# B&R Automation Studio project x20ost (part 3)

#### bnrdirmodule.c
```c
/********************************************************************
 * COPYRIGHT -- Kontora
 ********************************************************************
 * Program: bnrmain
 * File: bnrlsens.c
 * Author: Abramenya
 * Created: January 19, 2009
 *******************************************************************/

#include "bnrdirmodule.h"
#ifdef _DEFAULT_INCLUDES
 #include <AsDefault.h>
#endif
#if MYSYSTEM_ID != 5
void CDirectionModule_Init(This,SDIRTABLE *pDirect,CMFlash *pFlash)
{
    DECLARE_SINGLE_OPEN(CDirectionModule)
	INT i,nCreated;
	BOOL blSerialize;
	BYTE bySensorType,byLen;
	CSensor *pSensor;
	CSmartSensor *pSmartSensor;
	CIdleSensor *pIdleSensor;
	CDigitalSensor *pDgSensor;
	SNSPARAMTABLE *sP;
	pT->m_pDirTable = pDirect;
	pT->m_pFlash = pFlash;
	pT->m_wSensorMode = 0;
	pT->m_pvInGate = pDirect->pvIn;
	pT->m_pvOutGate = pDirect->pvOut;
	pT->m_byDefSett = 0;
    #if MYSYSTEM_ID == 4
	pT->m_byAmInpGate = ((SDIGGATES*)pT->m_pvInGate)->byAmGate;
    #else
    pT->m_byAmInpGate = ((SINPUTGATE*)pT->m_pvInGate)->byAmInGate;
    #endif
	pT->m_wLayerMode  = 0x2;
	/*
	#if   MYSYSTEM_ID == 0
	 pT->m_wLayerMode  = 0x2;
	#elif MYSYSTEM_ID == 1
	 pT->m_wLayerMode  = 0x1;
	#elif MYSYSTEM_ID == 2
	 pT->m_wLayerMode  = 0x2;
	#elif MYSYSTEM_ID == 3
	 pT->m_wLayerMode  = 0x1a;
	#endif
	*/
	pT->m_blGetData = FALSE;
    #ifdef DEB_CDirectionModule
	Info("\n(%b)CDIRC::>Create Direction.",&pDirect->byDirectionID);
    #endif
	pT->m_byStatSnsConn = 0xff;
	pT->m_byDirectionID = pDirect->byDirectionID;
	pT->m_byAmSwitching = pDirect->byAmSwitching;
	pT->m_byDirectionCode = pDirect->byDirectionCode;
    New(sizeof(CSensor*)*pT->m_byAmSwitching,pT->m_pSensor);
	for (i=0;i<pT->m_byAmSwitching;i++)pT->m_pSensor[i]=0;
	for (nCreated=0;nCreated<=1;nCreated++)
	{
	if(nCreated)
	{
     #if MYSYSTEM_ID != 4
	 pT->SetInputGate(pT,pT->m_pvInGate);
     #endif
	 blSerialize = pT->Serialize(pT,FALSE);
	}
	for (i=0;i<pT->m_byAmSwitching;i++)
	{
	 bySensorType = pDirect->sSwitchTable[i].bySwitchCommand;
	 switch(bySensorType)
	 {
	    case SWC_CMD_SMR_CON:
			{
			 if(nCreated==0){
			 New(sizeof(CSmartSensor),pSmartSensor);
			 InitObject(CSmartSensor,pSmartSensor);
			 pSmartSensor->pBase->m_bySystemID = pT->m_bySystemID;
			 pT->m_pSensor[i] = pSmartSensor->pBase;}
			 if(nCreated==1){
			 pSmartSensor->pBase = pT->m_pSensor[i];
			 pT->SwitchSensor(pT,pSmartSensor->pBase,&pDirect->sSwitchTable[i]);
			 pSmartSensor->pBase->SetDirection(pSmartSensor->pBase,pT,pT->m_byDirectionID);
			 pSmartSensor->pBase->Init(pSmartSensor->pBase,&pDirect->sSwitchTable[i]);}
			}
		break;
		case SWC_CMD_IDL_CON:
			{
			 if(nCreated==0){
			 New(sizeof(CIdleSensor),pIdleSensor);
			 InitObject(CIdleSensor,pIdleSensor);
			 pIdleSensor->pBase->m_bySystemID = pT->m_bySystemID;
			 pT->m_pSensor[i] = pIdleSensor->pBase;}
			 if(nCreated==1){
			 pIdleSensor->pBase = pT->m_pSensor[i];
			 pT->SwitchSensor(pT,pIdleSensor->pBase,&pDirect->sSwitchTable[i]);
			 pIdleSensor->pBase->SetDirection(pIdleSensor->pBase,pT,pT->m_byDirectionID);
			 pIdleSensor->pBase->Init(pIdleSensor->pBase,&pDirect->sSwitchTable[i]);}
			}
		break;
		case SWC_CMD_EMT_CON:
			{
			 if(nCreated==0){
			 New(sizeof(CSensor),pSensor);
			 InitObject(CSensor,pSensor);
			 pSensor->m_bySystemID = pT->m_bySystemID;
			 pT->m_pSensor[i] = pSensor;}
			 if(nCreated==1){
			 pSensor->pBase = pT->m_pSensor[i];
			 pSensor->SetDirection(pSensor,pT,pT->m_byDirectionID);
			 pSensor->Init(pSensor,&pDirect->sSwitchTable[i]);}
			}
		break;
		case SWC_CMD_LOG_CON:
			{
			 if(nCreated==0){
			 New(sizeof(CDigitalSensor),pDgSensor);
			 InitObject(CDigitalSensor,pDgSensor);
			 pDgSensor->pBase->m_bySystemID = pT->m_bySystemID;
			 pT->m_pSensor[i] = pDgSensor->pBase;}
			 if(nCreated==1){
			 pDgSensor->pBase = pT->m_pSensor[i];
             pDgSensor->pBase->SetDirection(pDgSensor->pBase,pT,pT->m_byDirectionID);
			 pDgSensor->pBase->InitDigital(pDgSensor->pBase,&pDirect->sSwitchTable[i]);//Create In Out
			 pT->SwitchDigitalSensor(pT,pDgSensor->pBase,&pDirect->sSwitchTable[i]);}   //Connect In or Out
			}
		break;
		default:
		break;
	 }
	}
	}
    #if MYSYSTEM_ID != 4
	if (blSerialize)for(i=0;i<8;i++)if(pT->m_nST.m_wLayerMode&(1<<i))pT->SetCurentTank(pT,i);
    #endif
}
BOOL CDirectionModule_EventHandler(This,SMESSAGE *pMsg)
{
    DECLARE_SINGLE_OPEN(CDirectionModule)
	INT16 **pwData;
	CSensor *pSN;
	BYTE byParam;
    switch(pMsg->m_sbyFor)
	{
		case MDL_DIRMD:
			 switch(pMsg->m_sbyType)
			 {
			    case EV_DIRMD_SET_TANK_REQ:
	                 pT->SetCurentTank(pT,pMsg->m_sbySensor);
                     #ifdef DEB_CDirectionModule
					 Info("\n(%b)CDIRC::>(%b)(%b)SetTank.",&pT->m_bySystemID,&pT->m_byDirectionID,&pMsg->m_sbySensor);
                     #endif
				break;
				#if MYSYSTEM_ID != 4
			 	case EV_DIRMD_GET_PARAM_REQ:
					 if(pMsg->m_sbySensor<pT->m_byAmSwitching)
					 {
					  pSN = pT->m_pSensor[pMsg->m_sbySensor];
					  byParam = pMsg->m_sbyInfo[1];
					  pSN->GetParamTable(pSN,pMsg->m_sbyInfo[1]);
                      #ifdef DEB_CDirectionModule
					  Info("\n(%b)CDIRC::>(%b)(%b)GetParam.",&pT->m_bySystemID,&pT->m_byDirectionID,&pMsg->m_sbySensor);
                      #endif
					 }
				break;
				case EV_DIRMD_CONN_STAT_SNS_IND:
                     #ifdef DEB_CDirectionModule
					 Info("\n(%b)CDIRC::>(%b)(%b)Connect To Sensor.",&pT->m_bySystemID,&pT->m_byDirectionID,&pMsg->m_sbySensor);
                     #endif
					 pT->m_byStatSnsConn  = pMsg->m_sbySensor;
					 pT->m_byTypeTest     = 0;
					 if(pMsg->m_sbySensor<pT->m_byAmSwitching)
					 {
					  pSN = pT->m_pSensor[pMsg->m_sbySensor];
					  pT->m_pStatSnsTmr.SetTimer(&pT->m_pStatSnsTmr,MDL_DIRMD,MDL_DIRMD,EV_DIRMD_REFR_TIM_PROC_IND,pSN->m_byDirection,0,DEV_SYSTM_BOX_ID);
					  pSN->GetParamTable(pSN,MDL_TPIDT);
					 }
				break;
			    case EV_DIRMD_DISC_STAT_SNS_IND:
                     #ifdef DEB_CDirectionModule
					 Info("\n(%b)CDIRC::>(%b)Disconnect To Sensor.",&pT->m_bySystemID,&pT->m_byDirectionID);
                     #endif
					 pT->m_byStatSnsConn = 0xff;
				break;
                #endif
			    case EV_DIRMD_CONN_STAT_START_IND:
                     #ifdef DEB_CDirectionModule
					 Info("\n(%b)CDIRC::>(%b)(%b)Start Stat Proc:%b.",&pT->m_bySystemID,&pT->m_byDirectionID,&pMsg->m_sbySensor,&pMsg->m_sbyInfo[1]);
                     #endif
					 if((pMsg->m_sbySensor<pT->m_byAmSwitching)&&(pT->m_byStatSnsConn!=0xff))
					 {
					  pSN = pT->m_pSensor[pMsg->m_sbySensor];
					  pT->m_byTypeTest = pMsg->m_sbyInfo[2];
					  if(pT->m_byTypeTest==0)pSN->StartCaptureProc(pSN);
					  pT->m_pStatSnsTmr.OnTimer(&pT->m_pStatSnsTmr,pMsg->m_sbyInfo[1]*SYSTEM_QTIME/100);
					 }
				break;
			    case EV_DIRMD_CONN_STAT_STOP_IND:
                     #ifdef DEB_CDirectionModule
					 Info("\n(%b)CDIRC::>(%b)(%b)Stop Stat Proc.",&pT->m_bySystemID,&pT->m_byDirectionID,&pMsg->m_sbySensor);
                     #endif
					 if(pMsg->m_sbySensor<pT->m_byAmSwitching)
					 {
					  pSN = pT->m_pSensor[pMsg->m_sbySensor];
 					  pT->m_pStatSnsTmr.OfTimer(&pT->m_pStatSnsTmr);
					 }
			    break;
				case EV_DIRMD_REFR_TIM_PROC_IND:
					 if(pT->m_byStatSnsConn!=0xff)
					 {
					 pMsg->m_sbyFrom      = MDL_DIRMD;
					 pMsg->m_sbyFor       = MDL_TPIDT;
					 pMsg->m_sbyIntType   = DEV_ARM_PORT_TCP;
					 pMsg->m_sbyServerID  = pT->m_bySystemID;
					 pMsg->m_sbyType      = EV_DIRMD_STAT_DATA_IND;
					 pMsg->m_sbyDirection = pT->m_byDirectionID;
	                 pMsg->m_sbySensor    = pT->m_byStatSnsConn;
 				     pSN                  = pT->m_pSensor[pT->m_byStatSnsConn];
                     if(pT->m_byTypeTest==0)
					 {
					  pMsg->m_sbyInfo[0] = (BYTE)pSN->m_wStatIndex;
					  pMsg->m_sbyInfo[1] = (BYTE)pSN->m_wStatIndex;
					  pwData = pSN->GetCaptureBuffer(pSN);
					  memcpy(&pMsg->m_sbyInfo[2],pwData,12*pSN->m_wStatQuant);
					  pMsg->m_swLen = 9+1+1+12*pSN->m_wStatQuant;
					 }
					 if(pT->m_byTypeTest==1)
					 {
					  pSN->CaptureData(pSN->pChld);
					  pwData = pSN->GetCaptureBuffer(pSN);
					  pMsg->m_sbyInfo[0] = (BYTE)pSN->m_wStatIndex;
					  pMsg->m_sbyInfo[1] = (BYTE)pSN->m_wStatIndex;
					  memcpy(&pMsg->m_sbyInfo[2],pwData,4*pSN->m_wStatIndex);
					  pMsg->m_swLen = 9+1+1+4*pSN->m_wStatIndex;
					 }
					 FPUT(DEV_ARMOT_BOX_ID,(BYTE*)&pMsg->m_swLen);
                     if(dwFL&DEB_OUT_OBSR_COMM)
	                 Info("\n(%b)COBSE::>msg:%M",&pT->m_bySystemID,(BYTE*)pMsg);
					 pSN->RestartCaptureProc(pSN);
					 pT->m_pStatSnsTmr.Restart(&pT->m_pStatSnsTmr);
					 }
				break;
			    default:
			    break;
			 }
		break;
		default:
		break;
	}
	return TRUE;
}
void CDirectionModule_SetInputGate(This,SINPUTGATE *pING)
{
    DECLARE_SINGLE_OPEN(CDirectionModule)
	REAL Imin,Imax,R;
	BYTE i;
	CSlot *pSL;
	CPin  *pPN;
	for (i=0;i<pT->m_byAmInpGate;i++)
	{
	 pSL = pT->m_pComputer->GetSlot(pT->m_pComputer,pING->mIn[i].bySrcSlotNumber);
     pPN = pSL->GetPin(pSL->pChld,pING->mIn[i].bySrcPinNumber);
	 InitObject(CInputGate,&pT->m_nInpGate[i]);
	 pT->m_nInpGate[i].Init(&pT->m_nInpGate[i],i,pPN->GetAddrPin(pPN->pChld),500.0,pING->mIn[i].m_swResistance);
	 #ifdef MY_MODEL
	 pT->m_pSensor[0]->m_sPT.m_swHiLimit = pING->mIn[i].m_swHiLimit;
	 pT->m_nInpGate[i].SetInput(&pT->m_nInpGate[i],pT->m_pSensor[0]->GetInParam(pT->m_pSensor[0],pING->mIn[i].m_swInitValue)/pT->m_nInpGate[i].m_rKoef);
     #endif
	}
}
void CDirectionModule_SwitchSensor(This,CSensor *pSensor,SSWITCHTABLE *pSwitchTable)
{
    DECLARE_SINGLE_OPEN(CDirectionModule)
	BYTE i;
	CSlot *pSL;
	CPin  *pPN;
	SOUTGATE *sG;
	COutGate *pGate;
	SNSPARAMTABLE *sP = (SNSPARAMTABLE*)pSwitchTable->sSensorParamTable;
	BYTE byOutState = sP->m_sbyOutState;
	pSensor->ConnectFCP(pSensor,&pT->m_nInpGate[sP->m_byID]);
	pSensor->m_byAmOutGate = pSwitchTable->byAmOutGate;
    for (i=0;i<pSwitchTable->byAmOutGate;i++)
    {
	  New(sizeof(COutGate),pGate);
	  InitObject(COutGate,pGate);
	  sG = (SOUTGATE*)pSwitchTable->sOutGate[i];
	  pSL = pT->m_pComputer->GetSlot(pT->m_pComputer,sG->byOutSlotNumber);
	  pPN = pSL->GetPin(pSL->pChld,sG->byOutPinNumber);
	  pGate->Init(pGate,
		          sG->byID,
		          sG->byType,
		          sG->byOType,
		          sG->byMode,
                  sG->rMinRamp,
		          sG->rMaxRamp,
		          pPN,
		          sG->wLoLimit,
		          sG->wHiLimit,
		          sG->wCurrOpen,
		          byOutState,
                  sP->m_swMaxAcpInp,
				  sG->wOpenTime,
		          sG->chName);
	  pSensor->ConnectOutGate(pSensor,pGate);
    }
}
void CDirectionModule_SwitchDigitalSensor(This,CSensor *pSensor,SSWITCHTABLE *pSwitchTable)
{
    DECLARE_SINGLE_OPEN(CDirectionModule)
	BYTE i;
	CSlot *pSL;
	CPin  *pPN;
	CComputer *pCM = pT->m_pComputer;
	SDIGGATE  *pDIN = pSwitchTable->sSensorParamTable;
	SDIGGATE  *pDOT = pSwitchTable->sOutGate[0];
    for (i=0;i<pDIN->swAmpin;i++)
    {
	  pSL = pCM->GetSlot(pCM,pDIN->sPinGate[i].sbySlot);
	  pPN = pSL->GetPin(pSL->pChld,pDIN->sPinGate[i].sbyPin);
	  pSensor->m_pINP[i] = pPN;
	}
    for (i=0;i<pDOT->swAmpin;i++)
    {
	  pSL = pCM->GetSlot(pCM,pDOT->sPinGate[i].sbySlot);
	  pPN = pSL->GetPin(pSL->pChld,pDOT->sPinGate[i].sbyPin);
	  pSensor->m_pOUT[i] = pPN;
	}
	pSensor->ConnectPinAddres(pSensor);
}
void CDirectionModule_ConnectToAdmin(This,CAdmin *pAdmin)
{
    DECLARE_SINGLE_OPEN(CDirectionModule)
	pT->m_pAdmin = pAdmin;
}
_GLOBAL INT  inAmSens,wwLen;
WORD CDirectionModule_GetInOutData(This,SMESSAGE *pMsg)
{
    DECLARE_SINGLE_OPEN(CDirectionModule)
	INT i,wLen;
	CSensor *p;
	BYTE *pM,*pIT,*pOT,*pW;
    pMsg->m_sbyFrom      = MDL_DIRMD;
	pMsg->m_sbyFor       = MDL_ARMSY;
	pMsg->m_sbyIntType   = DEV_ARM_PORT_TCP;
	pMsg->m_sbyType      = EV_OBSRV_GET_INOUT_SDATA_IND;
	pMsg->m_sbyServerID  = pT->m_bySystemID;
	pMsg->m_sbyDirection = pT->m_byDirectionID;
	pMsg->m_sbySensor    = 0xff;
	pM    = &pMsg->m_sbyInfo[0];
	pM[0] = pT->m_byAmSwitching;
	pM[1] = 4;
	inAmSens = 0;
	for(i=0;i<pT->m_byAmSwitching;i++)
	{
	  p = pT->m_pSensor[i];
	  pIT = (BYTE*)&p->m_nInPin;
	  pOT = (BYTE*)&p->m_nOutPin;
	  inAmSens++;
      #ifndef WIN32
	  pM[2+4*i+1]   = pIT[0];
	  pM[2+4*i+0]   = pIT[1];
	  pM[2+4*i+2+1] = pOT[0];
	  pM[2+4*i+2+0] = pOT[1];
	  #else
	  pM[2+4*i+0]   = pIT[0];
	  pM[2+4*i+1]   = pIT[1];
	  pM[2+4*i+2+0] = pOT[0];
	  pM[2+4*i+2+1] = pOT[1];
	  #endif
	}
	wLen = 9+1+1+4*pT->m_byAmSwitching;
	#ifndef WIN32
	pIT   = (BYTE*)pMsg;
	pOT   = (BYTE*)&wLen;
	pIT[1] = pOT[0];
	pIT[0] = pOT[1];
    #endif
	return wLen;
}
void CDirectionModule_GetDirMode(This,SMESSAGE *pMsg)
{
    DECLARE_SINGLE_OPEN(CDirectionModule)
	BYTE i;
	WORD wState = 0;
	CSensor *p;
	BYTE *pM,*pW,*pW0;
    pMsg->m_sbyFrom      = MDL_DIRMD;
	pMsg->m_sbyFor       = MDL_ARMSY;
	pMsg->m_sbyIntType   = DEV_ARM_PORT_TCP;
	pMsg->m_sbyType      = EV_OBSRV_GET_MODE_IND;
	pMsg->m_sbyServerID  = pT->m_bySystemID;
	pMsg->m_sbyDirection = pT->m_byDirectionID;
	pMsg->m_sbySensor    = 0xff;
	pMsg->m_sbyInfo[0]   = pT->m_byAmSwitching;
	pMsg->m_sbyInfo[1]   = 2;
	pM = &pMsg->m_sbyInfo[2];
	for(i=0;i<pT->m_byAmSwitching;i++)
	{
	 p = pT->m_pSensor[i];
	 if(p->m_sPT.m_sbyMode==SNS_MD_AUTO)wState |= 1<<i;
	}
	pMsg->m_swLen = 9+1+1+2;
	pW  = (BYTE*)&wState;
    #ifndef WIN32
	pM[1] = pW[0];
	pM[0] = pW[1];
    #else
    memcpy(pM,pW,2);
    #endif
	FPUT(DEV_ARMOT_BOX_ID,(BYTE*)pMsg);
	//Info("\n(%b)CDIRC::>MOD:MSG:%M",&pT->m_bySystemID,(BYTE*)pMsg);
}
void CDirectionModule_SetDirMode(This,SMESSAGE *pMsg)
{
    DECLARE_SINGLE_OPEN(CDirectionModule)
	BYTE i;
	WORD wMode;
	CSensor *p;
	wMode  = pT->GetWordParam(pT,&pMsg->m_sbyInfo[2]);
	for(i=0;i<pT->m_byAmSwitching;i++)
	{
	 p = pT->m_pSensor[i];
     if(wMode&(1<<i))p->SetAutoMode(p);else p->SetManMode(p);
	}
}
DWORD CDirectionModule_GetDwordParam(This,BYTE *pbyParam)
{
    DECLARE_SINGLE_OPEN(CSensor)
	DWORD dwValue;
	BYTE *pR = (BYTE*)&dwValue;
    #ifndef WIN32
	pR[3] = pbyParam[0];
	pR[2] = pbyParam[1];
	pR[1] = pbyParam[2];
	pR[0] = pbyParam[3];
    #else
	memcpy(&dwValue,pbyParam,4);
	#endif
	return dwValue;
}
WORD CDirectionModule_GetWordParam(This,BYTE *pbyParam)
{
    DECLARE_SINGLE_OPEN(CSensor)
	WORD wValue;
	BYTE *pR = (BYTE*)&wValue;
    #ifndef WIN32
	pR[1] = pbyParam[0];
	pR[0] = pbyParam[1];
    #else
	memcpy(&wValue,pbyParam,2);
	#endif
	return wValue;
}
WORD CDirectionModule_GetDigMcData(This,SMESSAGE *pMsg)
{
    DECLARE_SINGLE_OPEN(CDirectionModule)
	INT i,j;
	WORD wLen,wOut;
	CSensor *p;
	BYTE *pM,*pIT,*pOT;
    pMsg->m_sbyFrom      = MDL_DIRMD;
	pMsg->m_sbyFor       = MDL_ARMSY;
	pMsg->m_sbyIntType   = DEV_ARM_PORT_TCP;
	pMsg->m_sbyType      = EV_OBSRV_GET_DMC_DATA_IND;
	pMsg->m_sbyServerID  = pT->m_bySystemID;
	pMsg->m_sbyDirection = pT->m_byDirectionID;
	pMsg->m_sbySensor    = 0xff;
	pM    = &pMsg->m_sbyInfo[0];
	pM[0] = pT->m_byAmSwitching;
	pM[1] = 8;
	wLen = 9+1+1;
	for(i=0;i<pT->m_byAmSwitching;i++)
	{
	 p = pT->m_pSensor[i];
	 pT->AddDword(pT,&wLen,((BYTE*)pMsg+wLen),(BYTE*)&p->m_dwInState);
	 pT->AddDword(pT,&wLen,((BYTE*)pMsg+wLen),(BYTE*)&p->m_dwOutState);
	}
	#ifndef WIN32
	pIT   = (BYTE*)pMsg;
	pOT   = (BYTE*)&wLen;
	pIT[1] = pOT[0];
	pIT[0] = pOT[1];
    #else
    pMsg->m_swLen = wLen;
    #endif
	return wLen;
}
WORD CDirectionModule_GetXWData(This,SMESSAGE *pMsg)
{
    DECLARE_SINGLE_OPEN(CDirectionModule)
	INT i;
	WORD wLen,wOut,wIN;
	WORD wState=0,wLoArarmLimit=0,wHiArarmLimit=0,wSensorAlarm=0;
	CSensor *p;
	COutGate *pG;
	CInputGate *pI;
	UINT nInput;
	BYTE *pM,*pIT,*pOT,k=0;
    pMsg->m_sbyFrom      = MDL_DIRMD;
	pMsg->m_sbyFor       = MDL_ARMSY;
	pMsg->m_sbyIntType   = DEV_ARM_PORT_TCP;
	pMsg->m_sbyType      = EV_OBSRV_GET_OUT_DATA_IND;
	pMsg->m_sbyServerID  = pT->m_bySystemID;
	pMsg->m_sbyDirection = pT->m_byDirectionID;
	pMsg->m_sbySensor    = 0xff;
	pM    = &pMsg->m_sbyInfo[0];
	pM[0] = pT->m_byAmInpGate;
	pM[1] = pT->m_byAmSwitching;
	wLen = 9+1+1;wIN = 9+1+1+2*pT->m_byAmInpGate+4*pT->m_byAmSwitching;
	for(i=0;i<pT->m_byAmInpGate;i++)
	{
	 pI = &pT->m_nInpGate[i];
	 nInput = pI->GetMInput(pI);
	 pT->AddWord(pT,&wLen,((BYTE*)pMsg+wLen),(BYTE*)&nInput);
	 nInput = pI->m_pInpValue;
	 if((nInput>32700)||(nInput<6000))wSensorAlarm |= 0x1<<i;
	}
	for(i=0;i<pT->m_byAmSwitching;i++)
	{
	 p = pT->m_pSensor[i];
	 pT->AddWord(pT,&wLen,((BYTE*)pMsg+wLen),(BYTE*)&p->m_iIPHiLimit);
	 pT->AddWord(pT,&wLen,((BYTE*)pMsg+wLen),(BYTE*)&p->m_iIPLoLimit);
	 pG = p->m_pOutGate[0]; pM[wIN-9+k++] = pG->GetPrcGate(pG);
	 if(abs(p->m_nInPin-p->m_iPHiLimit)<1000) wState |= 0x1<<i;
	 if(p->m_blAlmLoLevel) wLoArarmLimit |= 0x1<<i;
	 if(p->m_blAlmHiLevel) wHiArarmLimit |= 0x1<<i;
	}
    wLen+=k;
    pT->AddWord(pT,&wLen,((BYTE*)pMsg+wLen),(BYTE*)&wState);
	pT->AddWord(pT,&wLen,((BYTE*)pMsg+wLen),(BYTE*)&pT->m_wSensorMode);
	pT->AddWord(pT,&wLen,((BYTE*)pMsg+wLen),(BYTE*)&pT->m_wLayerMode);
	pT->AddWord(pT,&wLen,((BYTE*)pMsg+wLen),(BYTE*)&wLoArarmLimit);
	pT->AddWord(pT,&wLen,((BYTE*)pMsg+wLen),(BYTE*)&wHiArarmLimit);
	pT->AddWord(pT,&wLen,((BYTE*)pMsg+wLen),(BYTE*)&wSensorAlarm);
	#ifndef WIN32
	pIT   = (BYTE*)pMsg;
	pOT   = (BYTE*)&wLen;
	pIT[1] = pOT[0];
	pIT[0] = pOT[1];
    #else
    pMsg->m_swLen = wLen;
    #endif
	return wLen;
}
void CDirectionModule_AddDword(This,WORD *pwLen,BYTE *byMsg,BYTE *byParam)
{
    DECLARE_SINGLE_OPEN(CDirectionModule)
    #ifndef WIN32
    byMsg[3] = byParam[0];
    byMsg[2] = byParam[1];
    byMsg[1] = byParam[2];
    byMsg[0] = byParam[3];
    #else
    memcpy(byMsg,byParam,4);
    #endif
    *pwLen += 4;
}
void CDirectionModule_AddWord(This,WORD *pwLen,BYTE *byMsg,BYTE *byParam)
{
    DECLARE_SINGLE_OPEN(CDirectionModule)
    #ifndef WIN32
    byMsg[1] = byParam[0];
    byMsg[0] = byParam[1];
    #else
    memcpy(byMsg,byParam,2);
    #endif
    *pwLen += 2;
}
void CDirectionModule_WordXCHG(This,SMESSAGE *pMsg)
{
	DECLARE_SINGLE_OPEN(CDirectionModule)
    #ifndef WIN32
	BYTE byTmp,*pW = (BYTE*)pMsg;
	byTmp = pW[0];
	pW[0] = pW[1];
	pW[1] = byTmp;
    #endif
}
void CDirectionModule_EnableGetData(This,BOOL byState)
{
     DECLARE_SINGLE_OPEN(CDirectionModule)
	 pT->m_blGetData = byState;
}
void CDirectionModule_ObserveProc(This)
{
	DECLARE_SINGLE_OPEN(CDirectionModule)
	CSensor *p;INT i;
	for(i=0;i<pT->m_byAmSwitching;i++)
	{
	 p = pT->m_pSensor[i];
	 if (p->m_bySensorType!=SNS_EMPTY) p->ObserveProc(p);
	}
}
void CDirectionModule_ConnectToComputer(This,CComputer *pComputer)
{
    DECLARE_SINGLE_OPEN(CDirectionModule)
	pT->m_pComputer = pComputer;
}
//_GLOBAL INT nValue_0,nValue_1,nValue_2,nValue_3,nValue_4,nValue_5,nValue_6;
BOOL CDirectionModule_Serialize(This,BOOL blDir)
{
	DECLARE_SINGLE_OPEN(CDirectionModule)
	BOOL res = TRUE;
	if (blDir==TRUE) res = pT->SaveContenst(pT);
	if (blDir==FALSE)res = pT->LoadContenst(pT);
	return res;
}
BOOL CDirectionModule_SaveContenst(This)
{
    DECLARE_SINGLE_OPEN(CDirectionModule)
	BOOL res = TRUE;
	pT->SaveTable(pT,&pT->m_nCT);
	//nValue_0++;
	if (!pT->m_pFlash->CompareMemory(pT->m_pFlash,(BYTE*)&pT->m_nCT,sizeof(SCONTENSTTABLE)))
	{
	 //nValue_1++;
	 //if (!pT->m_pFlash->WriteFlash(pT->m_pFlash,(BYTE*)&pT->m_nCT,sizeof(SCONTENSTTABLE)))
     if (!pT->m_pFlash->WriteFlashRem(pT->m_pFlash,(BYTE*)&pT->m_nCT,sizeof(SCONTENSTTABLE)))
	 {
	 	//nValue_2++;
		res = FALSE;
	 }
	}
	return res;
}
BOOL CDirectionModule_LoadContenst(This)
{
    DECLARE_SINGLE_OPEN(CDirectionModule)
	BOOL res = FALSE;
	pT->m_nST.m_bySystemID = 0xff;
	if (pT->m_pFlash->ReadFlash(pT->m_pFlash,(BYTE*)&pT->m_nST,sizeof(SCONTENSTTABLE)))
	{
	 if(pT->m_nST.m_byDefInit==1) return FALSE;
	 if(pT->m_nST.m_byDefInit==0)
	 {
	  if (pT->m_nST.m_bySystemID==pT->m_bySystemID)
	  {
      pT->LoadTable(pT,&pT->m_nST);
	  res = TRUE;
	  }
	 }
	}
	return res;
}
void CDirectionModule_SaveTable(This,SCONTENSTTABLE *psTable)
{
    DECLARE_SINGLE_OPEN(CDirectionModule)
	BYTE i;
	COutGate *pG;
	memset(psTable,0,sizeof(SCONTENSTTABLE));
	#if MYSYSTEM_ID != 4
	psTable->sInGate.byAmInGate   = pT->m_byAmInpGate;
	psTable->sOutGate.byAmOutGate = pT->m_byAmSwitching;
	psTable->m_byDefInit          = pT->m_byDefSett;
	for(i=0;i<pT->m_byAmInpGate;i++) psTable->mInResistance[i] = pT->m_nInpGate[i].m_rCurrRes;
	for(i=0;i<pT->m_byAmSwitching;i++)
	{
     memcpy(&psTable->sInGate.mIn[i],&pT->m_pSensor[i]->m_sPT,sizeof(SNSPARAMTABLE));
	 memcpy(&psTable->sOutGate.mOut[i],&pT->m_pSensor[i]->m_sGT,sizeof(SOUTGATE));
	 pG = pT->m_pSensor[i]->m_pOutGate[0];
	 psTable->sOutGate.mOut[i].wCurrOpen = pG->GetPrcGate(pG);
	 psTable->m_bySystemID = pT->m_bySystemID;
	}
	psTable->m_wLayerMode = pT->m_wLayerMode;
    #else
	psTable->m_bySystemID = pT->m_bySystemID;
    for(i=0;i<pT->m_byAmSwitching;i++) psTable->m_dwOutState[i] = pT->m_pSensor[i]->m_dwOutState;
    #endif
}
void CDirectionModule_LoadTable(This,SCONTENSTTABLE *psTable)
{
    DECLARE_SINGLE_OPEN(CDirectionModule)
	BYTE i;
	pT->m_byDefSett = psTable->m_byDefInit;
	#if MYSYSTEM_ID != 4
	for(i=0;i<pT->m_byAmInpGate;i++) pT->m_nInpGate[i].SetResistance(&pT->m_nInpGate[i],psTable->mInResistance[i]);
	for(i=0;i<pT->m_byAmSwitching;i++)
	{
	 pT->m_pDirTable->sSwitchTable[i].sSensorParamTable = &psTable->sInGate.mIn[i];
	 pT->m_pDirTable->sSwitchTable[i].sOutGate[0]       = &psTable->sOutGate.mOut[i];
	}
    #else
	for(i=0;i<pT->m_byAmSwitching;i++) pT->m_pSensor[i]->m_dwOutState = psTable->m_dwOutState[i];
    #endif
}
void CDirectionModule_SetCurentTank(This,BYTE byTank)
{
    DECLARE_SINGLE_OPEN(CDirectionModule)
	if(pT->m_bySystemID==3)
	{
	 if((byTank>=0)&&(byTank<=1))
	 {
	  pT->m_wLayerMode &= 0xfc;
	  pT->m_pSensor[0]->m_nInp = &pT->m_nInpGate[byTank];
	  pT->m_pSensor[0]->m_sPT.m_swResistance = pT->m_nInpGate[byTank].m_rCurrRes;
	 }
	 if((byTank>=2)&&(byTank<=3))
	 {
	  pT->m_wLayerMode &= 0xf3;
	  pT->m_pSensor[1]->m_nInp = &pT->m_nInpGate[byTank];
	  pT->m_pSensor[1]->m_sPT.m_swResistance = pT->m_nInpGate[byTank].m_rCurrRes;
	 }
 	 if((byTank>=4)&&(byTank<=7))
	 {
	  pT->m_wLayerMode &= 0x0f;
	  pT->m_pSensor[2]->m_nInp = &pT->m_nInpGate[byTank];
	  pT->m_pSensor[3]->m_nInp = &pT->m_nInpGate[byTank];
	  pT->m_pSensor[2]->m_sPT.m_swResistance = pT->m_nInpGate[byTank].m_rCurrRes;
	  pT->m_pSensor[3]->m_sPT.m_swResistance = pT->m_nInpGate[byTank].m_rCurrRes;
	 }
	}else
	{
	  pT->m_wLayerMode = 0;
	  pT->m_pSensor[0]->m_nInp = &pT->m_nInpGate[byTank];
	  pT->m_pSensor[1]->m_nInp = &pT->m_nInpGate[byTank];
	  pT->m_pSensor[0]->m_sPT.m_swResistance = pT->m_nInpGate[byTank].m_rCurrRes;
	  pT->m_pSensor[1]->m_sPT.m_swResistance = pT->m_nInpGate[byTank].m_rCurrRes;
	}
	pT->m_wLayerMode |= 1<<byTank;
}
void CDirectionModule_CDirectionModule(This)
{
    DECLARE_SINGLE_OPEN(CDirectionModule)
	DECLARE_REGISTRATION(CDirectionModule,Init)
	DECLARE_REGISTRATION(CDirectionModule,ConnectToComputer)
	DECLARE_REGISTRATION(CDirectionModule,SwitchSensor)
	DECLARE_REGISTRATION(CDirectionModule,ObserveProc)
	DECLARE_REGISTRATION(CDirectionModule,GetInOutData)
	DECLARE_REGISTRATION(CDirectionModule,EnableGetData)
	DECLARE_REGISTRATION(CDirectionModule,ConnectToAdmin)
	DECLARE_REGISTRATION(CDirectionModule,EventHandler)
	DECLARE_REGISTRATION(CDirectionModule,WordXCHG)
	DECLARE_REGISTRATION(CDirectionModule,GetXWData)
	DECLARE_REGISTRATION(CDirectionModule,GetDirMode)
	DECLARE_REGISTRATION(CDirectionModule,SetDirMode)
	DECLARE_REGISTRATION(CDirectionModule,GetDwordParam)
	DECLARE_REGISTRATION(CDirectionModule,GetWordParam)
	DECLARE_REGISTRATION(CDirectionModule,AddDword)
	DECLARE_REGISTRATION(CDirectionModule,AddWord)
	DECLARE_REGISTRATION(CDirectionModule,SwitchDigitalSensor)
	DECLARE_REGISTRATION(CDirectionModule,GetDigMcData)
	DECLARE_REGISTRATION(CDirectionModule,SetInputGate)
 	DECLARE_REGISTRATION(CDirectionModule,Serialize)
	DECLARE_REGISTRATION(CDirectionModule,SaveContenst)
	DECLARE_REGISTRATION(CDirectionModule,LoadContenst)
	DECLARE_REGISTRATION(CDirectionModule,SaveTable)
	DECLARE_REGISTRATION(CDirectionModule,LoadTable)
	DECLARE_REGISTRATION(CDirectionModule,SetCurentTank)
	InitObject(CMTimer,&pT->m_pStatSnsTmr);
	pT->m_pStatSnsTmr.SetTimer(&pT->m_pStatSnsTmr,MDL_DIRMD,MDL_DIRMD,EV_DIRMD_REFR_TIM_PROC_IND,0,0,DEV_SYSTM_BOX_ID);
}
void CDirectionModule_DCDirectionModule(This)
{
	DECLARE_SINGLE_OPEN(CDirectionModule)
	BYTE i,byType;
	for (i=0;i<pT->m_byAmSwitching;i++)
	{
	 byType = pT->m_pSensor[i]->m_bySwitchCommand;
	 if(byType==SWC_CMD_SMR_CON)DestroyObject(CSmartSensor,pT->m_pSensor[i]->pChld);
	 if(byType==SWC_CMD_IDL_CON)DestroyObject(CIdleSensor,pT->m_pSensor[i]->pChld);
	 if(byType==SWC_CMD_EMT_CON)DestroyObject(CSensor,pT->m_pSensor[i]);
	 if(byType==SWC_CMD_LOG_CON)DestroyObject(CDigitalSensor,pT->m_pSensor[i]->pChld);
	}
	Delete(sizeof(CSensor*)*pT->m_byAmSwitching,pT->m_pSensor);
}
DECLARE_SINGLE_CREATE(CDirectionModule)
#endif
```

#### bnrflash.c
```c
/********************************************************************
 * COPYRIGHT -- Kontora
 ********************************************************************
 * Program: bnrmain
 * File: bnrlsens.c
 * Author: Abramenya
 * Created: January 19, 2009
 *******************************************************************/

#include "bnrflash.h"
#ifdef _DEFAULT_INCLUDES
 #include <AsDefault.h>
#endif
#ifdef WIN32
SCONTENSTTABLE nMemory;
HANDLE hMFile;
void DMstore(struct DMstore* inst)
{
	DWORD dwBytesWritten;
	inst->status = 1;
	if(WriteFile(hMFile, (BYTE*)inst->data, sizeof(SCONTENSTTABLE),&dwBytesWritten, NULL))
	{
	 SetFilePointer(hMFile,0,NULL,FILE_BEGIN);
	 inst->status = 0;
	}
};
void DMxfree(struct DMxfree* inst){};
void DMfree(struct DMfree* inst){};
void DMxclear(struct DMxclear* inst){};
void DMclear(struct DMclear* inst){};
void DatObjCreate(struct DatObjCreate* inst){};
void DatObjWrite(struct DatObjWrite* inst){};
void DatObjRead(struct DatObjRead* inst)
{
     DWORD dwBytesWritten;
	 inst->status = 1;
	 if(ReadFile(hMFile, (BYTE*)inst->pDestination, inst->len,&dwBytesWritten, NULL))
	 {
      SetFilePointer(hMFile,0,NULL,FILE_BEGIN);
	  inst->status = 0;
	 }
};
void DatObjDelete(struct DatObjDelete* inst){};
void DatObjMove(struct DatObjMove* inst){};
void DatObjCopy(struct DatObjCopy* inst){};
void DatObjInfo(struct DatObjInfo* inst)
{
	inst->status = 0;
};
void DatObjChangeDate(struct DatObjChangeDate* inst){};
#endif
//DMstore_typ _GLOBAL DM_store_0;
BOOL CMFlash_WriteFlash(This,BYTE *pbyBuff,WORD wLen)
{
    DECLARE_SINGLE_OPEN(CMFlash)
	pT->ClearFlash(pT);
    pT->DM_store.enable   = 1;
    pT->DM_store.name     = (UDINT)pT->m_chName;
    pT->DM_store.data     = (UDINT)pbyBuff;
    pT->DM_store.size     = wLen;
    DMstore(&pT->DM_store);
	//memcpy(&DM_store_0,&pT->DM_store,sizeof(DMstore_typ));
    if (pT->DM_store.status == 0)return TRUE;
	else
	return FALSE;
}
BOOL CMFlash_WriteFlashRem(This,BYTE *pbyBuff,WORD wLen)
{
    DECLARE_SINGLE_OPEN(CMFlash)
	SLMESSAGE *pMsg;
    New(sizeof(SLMESSAGE),pMsg);
	pMsg->m_swLen        = 9+wLen;
    pMsg->m_sbyFrom      = MDL_OBSRV;
	pMsg->m_sbyFor       = MDL_ARMSY;
	pMsg->m_sbyIntType   = DEV_ARM_PORT_TCP;
	pMsg->m_sbyType      = EV_OBSRV_REMFLS_SAVE_REQ;
	pMsg->m_sbyServerID  = MYSYSTEM_ID;
	pMsg->m_sbyDirection = 0xff;
	pMsg->m_sbySensor    = 0xff;
	memcpy(pMsg->m_sbyInfo,pbyBuff,wLen);
	FPUT(DEV_ARMOT_BOX_ID,(BYTE*)pMsg);
    Delete(sizeof(SLMESSAGE),pMsg);
	return TRUE;
}
INT CMFlash_Free(This)
{
	DECLARE_SINGLE_OPEN(CMFlash)
	pT->DM_free.enable = 1;
    DMfree(&pT->DM_free);
	return pT->DM_free.size;
}
//INT _GLOBAL nVL0,nVL1,nVL2,nVL3,nVL4;
//UDINT _GLOBAL pAddr,pAddr_0;
BOOL CMFlash_ReadFlash(This,BYTE *pbyBuff,WORD wLen)
{
    DECLARE_SINGLE_OPEN(CMFlash)
	BOOL res = FALSE;
    pT->DOInfo.enable     = 1;
    pT->DOInfo.pName      = (UDINT)pT->m_chName;
    DatObjInfo(&pT->DOInfo);
	//memcpy(&DOInfo_0,&pT->DOInfo,sizeof(DatObjInfo_typ));
	//nVL3++;
    if (pT->DOInfo.status == 0)
	{
     pT->DORead.enable    = 1;
     pT->DORead.ident     = pT->DOInfo.ident;
     pT->DORead.Offset    = 0;
	 pT->DORead.pDestination = (UDINT)pbyBuff;
	 //pAddr = pT->DORead.pDestination;
     pT->DORead.len       = wLen;
     DatObjRead(&pT->DORead);
	 //memcpy(&DORead_0,&pT->DORead,sizeof(DatObjRead_typ));
	 //nVL4++;
     if (pT->DORead.status == 0)res = TRUE; else
	 res = FALSE;
	}
	return res;
}
//USINT _GLOBAL byGlBuff1[200],byGlBuff2[200];
//USINT *pbyBuff_1;
//UINT _GLOBAL status_m;
BOOL CMFlash_CompareMemory(This,BYTE *bySrc,WORD wLen)
{
    DECLARE_SINGLE_OPEN(CMFlash)
	BOOL res=TRUE;
	WORD i;
	BYTE *pbyBuff;
	New(wLen,pbyBuff);
	//pAddr_0 = pbyBuff;
	if (pT->ReadFlash(pT,pbyBuff,wLen))
	{
	 //nVL0++;
	 for(i=0;i<wLen;i++)
	 {
	  //if(i<200)
	  //{
	  // byGlBuff1[i] = bySrc[i];
	  // byGlBuff2[i] = pbyBuff[i];
	  //}
	 if(pbyBuff[i]!=bySrc[i])
	 {
	  //nVL1++;
	  res = FALSE;
	  break;
	  //Delete(wLen,pbyBuff);
	  //return FALSE;
	 }
	 }
	}else res = FALSE;
	Delete(wLen,pbyBuff);
    return res;
}
BOOL CMFlash_ClearFlash(This)
{
	DECLARE_SINGLE_OPEN(CMFlash)
	BOOL res = TRUE;
	pT->DM_clear.enable = 1;
	DMclear(&pT->DM_clear);
	if (pT->DM_clear.status != 0) res = FALSE;
	return res;
}
void CMFlash_CMFlash(This)
{
    DECLARE_SINGLE_OPEN(CMFlash)
	DECLARE_REGISTRATION(CMFlash,WriteFlash)
	DECLARE_REGISTRATION(CMFlash,WriteFlashRem)
	DECLARE_REGISTRATION(CMFlash,ReadFlash)
	DECLARE_REGISTRATION(CMFlash,CompareMemory)
	DECLARE_REGISTRATION(CMFlash,ClearFlash)
	DECLARE_REGISTRATION(CMFlash,Free)
	pT->m_byFirstBlock    = 1;
	pT->m_byAmBlock       = 1;
	strcpy(pT->m_chName,"FlashModule");
    #ifdef WIN32
	hMFile = CreateFile("mflash.fls",
		GENERIC_READ|GENERIC_WRITE,
		FILE_SHARE_READ|FILE_SHARE_WRITE,
		NULL,
		OPEN_ALWAYS,
		FILE_ATTRIBUTE_NORMAL,
		NULL);
    #endif
	memset(&pT->DM_free,0,sizeof(DMfree_typ));
	memset(&pT->DM_clear,0,sizeof(DMclear_typ));
	memset(&pT->DM_store,0,sizeof(DMstore_typ));
}
void CMFlash_DCMFlash(This)
{
	DECLARE_SINGLE_OPEN(CMFlash)
}
DECLARE_SINGLE_CREATE(CMFlash)
```

#### bnrhardpin.c
```c
/********************************************************************
 * COPYRIGHT -- Kontora
 ********************************************************************
 * Program: bnrmain
 * File: bnrlsens.c
 * Author: Abramenya
 * Created: January 19, 2009
 *******************************************************************/

#include "bnrhardpin.h"
#ifdef _DEFAULT_INCLUDES
 #include <AsDefault.h>
#endif
//Analog Pin
void CAnalogPin_InitPin(This,PVOID pValue)
{
     DECLARE_MULTI_OPEN(CAnalogPin,CPin)
	 pT->m_vpHardPin = (UINT*)pValue;
}
void CAnalogPin_SetPin(This,SPIN *pPin)
{
     DECLARE_MULTI_OPEN(CAnalogPin,CPin)
	 *pT->m_vpHardPin = pPin->iValue;
}
void CAnalogPin_GetPin(This,SPIN *pPin)
{
     DECLARE_MULTI_OPEN(CAnalogPin,CPin)
	 pPin->iValue = *pT->m_vpHardPin;
}
PVOID CAnalogPin_GetAddrPin(This)
{
	 DECLARE_MULTI_OPEN(CAnalogPin,CPin)
	 return (PVOID)pT->m_vpHardPin;
}
void CAnalogPin_CAnalogPin(This)
{
     DECLARE_MULTI_OPEN(CAnalogPin,CPin)
	 DECLARE_VIRTUAL_FUNC(CAnalogPin,InitPin)
	 DECLARE_VIRTUAL_FUNC(CAnalogPin,GetPin)
	 DECLARE_VIRTUAL_FUNC(CAnalogPin,SetPin)
	 DECLARE_VIRTUAL_FUNC(CAnalogPin,GetAddrPin)
}
void CAnalogPin_DCAnalogPin(This)
{
	 DECLARE_MULTI_OPEN(CAnalogPin,CPin)
}
DECLARE_MULTI_CREATE(CAnalogPin,CPin)
//Digital Pin
void CDigitalPin_InitPin(This,PVOID pValue)
{
	 DECLARE_MULTI_OPEN(CDigitalPin,CPin)
	 pT->m_vpHardPin = (BOOL*)pValue;
}
void CDigitalPin_SetPin(This,SPIN *pPin)
{
 	 DECLARE_MULTI_OPEN(CDigitalPin,CPin)
	 *pT->m_vpHardPin = pPin->blValue;
}
void CDigitalPin_GetPin(This,SPIN *pPin)
{
	 DECLARE_MULTI_OPEN(CDigitalPin,CPin)
	 pPin->blValue = *pT->m_vpHardPin;
}
PVOID CDigitalPin_GetAddrPin(This)
{
	 DECLARE_MULTI_OPEN(CDigitalPin,CPin)
	 return pT->m_vpHardPin;
}
void CDigitalPin_CDigitalPin(This)
{
     DECLARE_MULTI_OPEN(CDigitalPin,CPin)
	 DECLARE_VIRTUAL_FUNC(CDigitalPin,InitPin)
	 DECLARE_VIRTUAL_FUNC(CDigitalPin,GetPin)
	 DECLARE_VIRTUAL_FUNC(CDigitalPin,SetPin)
	 DECLARE_VIRTUAL_FUNC(CDigitalPin,GetAddrPin)
}
void CDigitalPin_DCDigitalPin(This)
{
	 DECLARE_MULTI_OPEN(CDigitalPin,CPin)
}
DECLARE_MULTI_CREATE(CDigitalPin,CPin)
//Counter Pin
void CDCounterPin_InitPin(This,PVOID pValue)
{
	 DECLARE_MULTI_OPEN(CDCounterPin,CPin)
		pT->m_vpHardPin = (UINT*)pValue;
}
void CDCounterPin_SetPin(This,SPIN *pPin)
{
	 DECLARE_MULTI_OPEN(CDCounterPin,CPin)
		*pT->m_vpHardPin = pPin->blValue;
}
void CDCounterPin_GetPin(This,SPIN *pPin)
{
	 DECLARE_MULTI_OPEN(CDCounterPin,CPin)
		pPin->blValue = *pT->m_vpHardPin;
}
PVOID CDCounterPin_GetAddrPin(This)
{
	 DECLARE_MULTI_OPEN(CDCounterPin,CPin)
		return pT->m_vpHardPin;
}
void CDCounterPin_CDCounterPin(This)
{
	 DECLARE_MULTI_OPEN(CDCounterPin,CPin)
	 DECLARE_VIRTUAL_FUNC(CDCounterPin,InitPin)
	 DECLARE_VIRTUAL_FUNC(CDCounterPin,GetPin)
	 DECLARE_VIRTUAL_FUNC(CDCounterPin,SetPin)
	 DECLARE_VIRTUAL_FUNC(CDCounterPin,GetAddrPin)
}
void CDCounterPin_DCDCounterPin(This)
{
	 DECLARE_MULTI_OPEN(CDCounterPin,CPin)
}
DECLARE_MULTI_CREATE(CDCounterPin,CPin)
//Temperature Pin
void CTemperaturePin_InitPin(This,PVOID pValue)
{
	DECLARE_MULTI_OPEN(CTemperaturePin,CPin)
	pT->m_vpHardPin = (UINT*)pValue;
}
void CTemperaturePin_SetPin(This,SPIN *pPin)
{
	DECLARE_MULTI_OPEN(CTemperaturePin,CPin)
	*pT->m_vpHardPin = pPin->blValue;
}
void CTemperaturePin_GetPin(This,SPIN *pPin)
{
	DECLARE_MULTI_OPEN(CTemperaturePin,CPin)
	pPin->blValue = *pT->m_vpHardPin;
}
PVOID CTemperaturePin_GetAddrPin(This)
{
	DECLARE_MULTI_OPEN(CTemperaturePin,CPin)
	return pT->m_vpHardPin;
}
void CTemperaturePin_CTemperaturePin(This)
{
	DECLARE_MULTI_OPEN(CTemperaturePin,CPin)
	DECLARE_VIRTUAL_FUNC(CTemperaturePin,InitPin)
	DECLARE_VIRTUAL_FUNC(CTemperaturePin,GetPin)
	DECLARE_VIRTUAL_FUNC(CTemperaturePin,SetPin)
	DECLARE_VIRTUAL_FUNC(CTemperaturePin,GetAddrPin)
}
void CTemperaturePin_DCTemperaturePin(This)
{
	DECLARE_MULTI_OPEN(CTemperaturePin,CPin)
}
DECLARE_MULTI_CREATE(CTemperaturePin,CPin)
```

#### bnrhconfig.c
```c
#include "bnrhconfig.h"
#if MYSYSTEM_ID == 5
//Признак аварийности
AI_ASVL(0)
AI_ASVL(1)
AI_ASVL(2)
AI_ASVL(3)

AI_ASVL(4)
AI_ASVL(5)

AO_ASVL(6)

DI_ASVL(7)
DI_ASVL(8)

/*
DI_ASVL(9)
DI_ASVL(10)
DI_ASVL(11)
DI_ASVL(12)
DI_ASVL(13)
DI_ASVL(14)
DI_ASVL(15)
DI_ASVL(16)
DI_ASVL(17)
*/
DO_ASVL(9)
DO_ASVL(10)

//Подключение переменных по авариям
AIP2_ALVL(4) /**/ AI2_ALSL(4)
AIP2_ALVL(5) /**/ AI2_ALSL(5)

AOP4_ALVL(6)  /**/ AO4_ALSL(6)

DIP12_ALVL(7) /**/ DI12_ALSL(7)
DIP12_ALVL(8) /**/ DI12_ALSL(8)

//DIP2_ALVL(9)  /**/ DI2_ALSL(9)
//DIP2_ALVL(10) /**/ DI2_ALSL(10)
//DIP2_ALVL(11) /**/ DI2_ALSL(11)
//DIP2_ALVL(12) /**/ DI2_ALSL(12)
//DIP2_ALVL(13) /**/ DI2_ALSL(13)
//DIP2_ALVL(14) /**/ DI2_ALSL(14)
//DIP2_ALVL(15) /**/ DI2_ALSL(15)
//DIP2_ALVL(16) /**/ DI2_ALSL(16)
//DIP2_ALVL(17) /**/ DI2_ALSL(17)

DOP12_ALVL(9) /**/ DO12_ALSL(9)
DOP12_ALVL(10) /**/ DO12_ALSL(10)

//Инициализация информационных переменных
//AI
AIP2_AVL(4)  /**/ AI2_SL(4)
AIP2_AVL(5)  /**/ AI2_SL(5)
AOP4_AVL(6)  /**/ AO4_SL(6)
//DI
DIP12_AVL(7) /**/ DI12_SL(7)
DIP12_AVL(8) /**/ DI12_SL(8)

//DIP2_AVL(9)  /**/ DIC2_SL(9)
//DIP2_AVL(10) /**/ DIC2_SL(10)
//DIP2_AVL(11) /**/ DIC2_SL(11)
//DIP2_AVL(12) /**/ DIC2_SL(12)
//DIP2_AVL(13) /**/ DIC2_SL(13)
//DIP2_AVL(14) /**/ DIC2_SL(14)
//DIP2_AVL(15) /**/ DIC2_SL(15)
//DIP2_AVL(16) /**/ DIC2_SL(16)
//DIP2_AVL(17) /**/ DIC2_SL(17)
//DO
DOP12_AVL(9)  /**/ DO12_SL(9)
DOP12_AVL(10) /**/ DO12_SL(10)
#endif
#if MYSYSTEM_ID == 5
SKPPARAM nKP = {0,0,1,20,"Password","+375291415925","+000000000000","+000000000000"};
/*
typedef struct _tagArmInterface
{
BYTE byNumber;
BYTE byType;
BYTE byPortRate;
BYTE byAmTCPPort;
DWORD dwpPortNumber[DEV_MAX_TCP_PORT];
STCPADDR stTcpAddr;
}SARMINTERFACE;
*/
SARMINTERFACE nARM0   = {0,DEV_ARM_PORT_COM232,DEV_ARM_RATE_57600,0,{0    ,    0},{  EVEN,   D_8,  S_1,  0}};
SARMINTERFACE nARM1   = {1,DEV_ARM_PORT_COM232,DEV_ARM_RATE_9600,0 ,{0    ,    0},{  NOPAR,  D_8,  S_1,  0}};
SARMINTERFACE nARM2   = {2,DEV_ARM_PORT_COM232,DEV_ARM_RATE_9600,0 ,{0    ,    0},{  NOPAR,  D_8,  S_1,  0}};

SARMINTERFACE nARMTCP = {3,DEV_ARM_PORT_TCP,DEV_ARM_RATE_57600,0,{20001   ,20001},{  192,  168,  1,  4},"192.168.1.4"};
SARMINTERFACE nARMUDP = {4,DEV_ARM_PORT_UDP,DEV_ARM_RATE_100MB,0,{20003   ,20002},{  192,  168,  1,  5},"192.168.1.5"};

SHARDCOMPUTERTABLE nConfigTable =
{
	DEV_CPU_TYPE_X20,MYSYSTEM_ID,"Motorola m68 PS794","Version: Wather St","Date:15.02.2013",11,5,
		&nKP,
	{
		{&nARM0},{&nARM1},{&nARM2},{&nARMTCP},{&nARMUDP},
	},
	{
		{0  ,DEV_PLC_CPU_X20  ,                       0,1,0,&blAsValueAI0, NULL         ,         NULL},
		{1  ,DEV_PWCOM_PS9500,                        0,1,0,&blAsValueAI1, NULL         ,         NULL},       //IF4.ST0
		{2  ,DEV_COM_CS1020,                          0,1,0,&blAsValueAI2, NULL         ,         NULL},       //IF4.ST1
		{3  ,DEV_COM_CS1020,                          0,1,0,&blAsValueAI3, NULL         ,         NULL},       //IF4.ST2

		{4  ,DEV_AI_X20AI2622 ,DEV_MAX_AI_X20AI2622_PIN,1,0,&blAsValueAI4, blpAlValueAI4,  uipValueAI4},       //IF4.ST3
		{5  ,DEV_AT_X20AT2222 ,DEV_MAX_AT_X20AT2222_PIN,1,0,&blAsValueAI5, blpAlValueAI5,  uipValueAI5},       //IF4.ST4

		{6  ,DEV_AO_X20AO4622 ,DEV_MAX_AI_X20AI4622_PIN,1,0,&blAsValueAO6, blpAlValueAO6,  uipValueAO6},       //IF4.ST5

		{7  ,DEV_DI_X20DI9371 ,DEV_MAX_DI_X20DI9371_PIN,1,0,&blAsValueDI7,blpAlValueDI7 , blpValueDI7},        //IF4.ST6
		{8  ,DEV_DI_X20DI9371 ,DEV_MAX_DI_X20DI9371_PIN,1,0,&blAsValueDI8,blpAlValueDI8 , blpValueDI8},        //IF4.ST7

		//{9  ,DEV_DI_X20DI2377 ,DEV_MAX_DI_X20DI2377_PIN,1,0,&blAsValueDI9,blpAlValueDI9 , uipValueDI9},
		//{10 ,DEV_DI_X20DI2377 ,DEV_MAX_DI_X20DI2377_PIN,1,0,&blAsValueDI10,blpAlValueDI10, uipValueDI10},
		//{11 ,DEV_DI_X20DI2377 ,DEV_MAX_DI_X20DI2377_PIN,1,0,&blAsValueDI11,blpAlValueDI11, uipValueDI11},
		//{12 ,DEV_DI_X20DI2377 ,DEV_MAX_DI_X20DI2377_PIN,1,0,&blAsValueDI12,blpAlValueDI12, uipValueDI12},
		//{13 ,DEV_DI_X20DI2377 ,DEV_MAX_DI_X20DI2377_PIN,1,0,&blAsValueDI13,blpAlValueDI13, uipValueDI13},
		//{14 ,DEV_DI_X20DI2377 ,DEV_MAX_DI_X20DI2377_PIN,1,0,&blAsValueDI14,blpAlValueDI14, uipValueDI14},
		//{15 ,DEV_DI_X20DI2377 ,DEV_MAX_DI_X20DI2377_PIN,1,0,&blAsValueDI15,blpAlValueDI15, uipValueDI15},
		//{16 ,DEV_DI_X20DI2377 ,DEV_MAX_DI_X20DI2377_PIN,1,0,&blAsValueDI16,blpAlValueDI16, uipValueDI16},
		//{17 ,DEV_DI_X20DI2377 ,DEV_MAX_DI_X20DI2377_PIN,1,0,&blAsValueDI17,blpAlValueDI17, uipValueDI17},

		{9  ,DEV_DO_X20DO9321 ,DEV_MAX_DO_X20DO9321_PIN,1,0,&blAsValueDO9 ,blpAlValueDO9 ,blpValueDO9},        //IF4.ST8
		{10 ,DEV_DO_X20DO9321 ,DEV_MAX_DO_X20DO9321_PIN,1,0,&blAsValueDO10,blpAlValueDO10,blpValueDO10},       //IF4.ST9
		}
};
#endif

void InitHardValue(void)
{
	BYTE i;
	//BOOL blV;
	#if MYSYSTEM_ID == 5
	blAsValueAI0  = TRUE;
    blAsValueAI1  = TRUE;
   	blAsValueAI2  = TRUE;
    blAsValueAI3  = TRUE;
    blAsValueAI4  = TRUE;
    blAsValueAI5  = TRUE;
    blAsValueAO6  = TRUE;

    blAsValueDI7  = TRUE;
    blAsValueDI8  = TRUE;

    //blAsValueDI9  = TRUE;
	//blAsValueDI10 = TRUE;
    //blAsValueDI11 = TRUE;
    //blAsValueDI12 = TRUE;
    //blAsValueDI13 = TRUE;
    //blAsValueDI14 = TRUE;
    //blAsValueDI16 = TRUE;
    //blAsValueDI17 = TRUE;

	blAsValueDO9 = TRUE;
    blAsValueDO10 = TRUE;

	AI2_ALCSL(4)   AI_ALIN2(4,FALSE)
	AI2_ALCSL(5)   AI_ALIN2(5,FALSE)
	AO4_ALCSL(6)   AO_ALOT4(6,FALSE)

    DI12_ALCSL(7) DI_ALIN12(7,FALSE)
	DI12_ALCSL(8) DI_ALIN12(8,FALSE)

	//DI2_ALCSL(9)  DI_ALIN2(9,FALSE)
	//DI2_ALCSL(10) DI_ALIN2(10,FALSE)
	//DI2_ALCSL(11) DI_ALIN2(11,FALSE)
	//DI2_ALCSL(12) DI_ALIN2(12,FALSE)
	//DI2_ALCSL(13) DI_ALIN2(13,FALSE)
	//DI2_ALCSL(14) DI_ALIN2(14,FALSE)
	//DI2_ALCSL(15) DI_ALIN2(15,FALSE)
	//DI2_ALCSL(16) DI_ALIN2(16,FALSE)
	//DI2_ALCSL(17) DI_ALIN2(17,FALSE)

	DO12_ALCSL(9)  DO_ALIN12(9,FALSE)
	DO12_ALCSL(10) DO_ALIN12(10,FALSE)

	//*blpAlValueAI2[0] = 1;
	//*blpAlValueAI2[byParam0] = byParam1;

	//blValueDO17_1 = 0;
	AI2_CSL(4)  /*Init*/
	AI2_CSL(5)  /*Init*/
	AO4_CSL(6)  /*Init*/

    DI12_CSL(7) /*Init*/DI_INI12(7,FALSE)
	DI12_CSL(8) /*Init*/DI_INI12(8,FALSE)

	//DIC2_CSL(9)  /*Init*/DIC_INI2(9,FALSE)
	//DIC2_CSL(10) /*Init*/DIC_INI2(10,FALSE)
	//DIC2_CSL(11) /*Init*/DIC_INI2(11,FALSE)
	//DIC2_CSL(12) /*Init*/DIC_INI2(12,FALSE)
	//DIC2_CSL(13) /*Init*/DIC_INI2(13,FALSE)
	//DIC2_CSL(14) /*Init*/DIC_INI2(14,FALSE)
	//DIC2_CSL(15) /*Init*/DIC_INI2(15,FALSE)
	//DIC2_CSL(16) /*Init*/DIC_INI2(16,FALSE)
	//DIC2_CSL(17) /*Init*/DIC_INI2(17,FALSE)

	DO12_CSL(9) /*Init*/
	DO12_CSL(10) /*Init*/
    #endif
}
```

#### bnridlesensor.c
```c
/********************************************************************
 * COPYRIGHT -- Kontora
 ********************************************************************
 * Program: bnrmain
 * File: bnrlsens.c
 * Author: Abramenya
 * Created: January 19, 2009
 *******************************************************************/

#include "bnridlesensor.h"
#if MYSYSTEM_ID != 5
#ifdef _DEFAULT_INCLUDES
 #include <AsDefault.h>
#endif
extern SINT *chSensType[];
extern SINT *chParType[];
void CIdleSensor_InitSensor(This,PVOID pvParam)
{
    DECLARE_MULTI_OPEN(CIdleSensor,CSensor)
	SNSPARAMTABLE *pParam = (SNSPARAMTABLE*)pvParam;
	pT->SetState(pT,TRUE);
    #ifdef DEB_CIdleSensor
	Info("\n(%b)CISNS::>Create SNS.:%s.:%s.Rng:[%w..%w].AlarmRng:[%w..%w]",
    &pB->m_bySensorID,
    chSensType[pB->m_bySensorType],
	chParType[pB->m_byParamType],
	&pB->m_iLoLimit,&pB->m_iHiLimit,
	&pB->m_iLoAlmLimit,&pB->m_iHiAlmLimit
	);
	#endif
}
void CIdleSensor_IncInput(This,INT16 wParam)
{
    DECLARE_MULTI_OPEN(CIdleSensor,CSensor)
	COutGate *pG0 = pB->m_pOutGate[0];
	pG0->SetGate(pG0,pB->m_nInPin);
	pB->m_nInPin += wParam;
	//Info("\n(%b)CIDSN::>DC(%b,%b)PR_INC::%w.",&pB->m_bySystemID,&pB->m_byDirection,&pB->m_bySensorID,&pB->m_sInPin.iValue);
}
void CIdleSensor_SetInput(This,SPIN *pValue)
{
    DECLARE_MULTI_OPEN(CIdleSensor,CSensor)
	COutGate *pG0 = pB->m_pOutGate[0];
	pB->m_nInPin = pValue->iValue;
	pG0->SetGate(pG0,pB->m_nInPin);
	//Info("\n(%b)CIDSN::>DC(%b,%b)PR_X::%w.",&pB->m_bySystemID,&pB->m_byDirection,&pB->m_bySensorID,&pB->m_sInPin.iValue);
}
void CIdleSensor_SetOutput(This,BYTE byNumber,SPIN *pValue)
{
	DECLARE_MULTI_OPEN(CIdleSensor,CSensor)
	COutGate *pG0 = pB->m_pOutGate[byNumber];
	pB->m_nOutPin = pValue->iValue;
	if(pG0)pG0->SetGate(pG0,pB->m_nOutPin);
}
void CIdleSensor_PreProc(This)
{
    DECLARE_MULTI_OPEN(CIdleSensor,CSensor)
	pB->m_nInPin = pB->m_nInp->GetInput(pB->m_nInp);
}
void CIdleSensor_Processing(This)
{
    DECLARE_MULTI_OPEN(CIdleSensor,CSensor)
}
void CIdleSensor_PostProc(This)
{
    DECLARE_MULTI_OPEN(CIdleSensor,CSensor)
}
void CIdleSensor_CaptureData(This)
{
	DECLARE_MULTI_OPEN(CIdleSensor,CSensor)
	INT16 wValue = 0;
	INT16 wValue1 = 0;
	COutGate *pG0 = pB->m_pOutGate[0];
	COutGate *pG1 = pB->m_pOutGate[1];
	if(pG0)wValue  = pG0->GetGate(pG0);
	if(pG1)wValue1 = pG1->GetGate(pG1);
	pB->OpenGate(pB);
	pB->AddData(pB,(DINT)pB->m_nInPin);
	pB->AddData(pB,(DINT)wValue1);
	pB->AddData(pB,(DINT)wValue);
	pB->AddData(pB,0);
	pB->AddData(pB,0);
	pB->AddData(pB,0);
	pB->AddData(pB,0);
	pB->CloseGate(pB);
}
BOOL CIdleSensor_GetState(This)
{
    DECLARE_MULTI_OPEN(CIdleSensor,CSensor)
	return pT->m_blState;
}
void CIdleSensor_SetState(This,BOOL blBool)
{
    DECLARE_MULTI_OPEN(CIdleSensor,CSensor)
	pT->m_blState = blBool;
}
void CIdleSensor_EventHandler(This,SMESSAGE *pMsg)
{
    DECLARE_MULTI_OPEN(CIdleSensor,CSensor)
	SPIN nPin;
	REAL rlParam;
	BYTE byLen,byInitType,byPType,byPLen,*pR=(BYTE*)&rlParam;
	switch(pMsg->m_sbyType)
	{
	  case EV_SMSNS_SET_PARAM_REQ:
		 byLen      = pMsg->m_sbyInfo[0];
		 byInitType = pMsg->m_sbyInfo[1];
		 byPType    = pMsg->m_sbyInfo[2];
		 byPLen     = pMsg->m_sbyInfo[3];
         #ifdef DEB_CIdleSensor
		 Info("\n(%b)CIDSN::>DC(%b,%b)SSP:%M.",&pB->m_bySystemID,&pB->m_byDirection,&pB->m_bySensorID,(BYTE*)pMsg);
         #endif
		 if(byInitType==SNS_SENS_INI)
		 {
		  if(byPType==PR_X)
		  {
			nPin.iValue = pB->GetWordParam(pB,&pMsg->m_sbyInfo[4]);
    		pT->SetInput(pT,&nPin);
		  }
		 }
	  break;
	  default:
	  break;
	};
}
void CIdleSensor_CIdleSensor(This)
{
    DECLARE_MULTI_OPEN(CIdleSensor,CSensor)
	DECLARE_REGISTRATION(CIdleSensor,SetState)
	DECLARE_REGISTRATION(CIdleSensor,GetState)
	DECLARE_VIRTUAL_FUNC(CIdleSensor,EventHandler)
	DECLARE_VIRTUAL_FUNC(CIdleSensor,SetInput)
	DECLARE_VIRTUAL_FUNC(CIdleSensor,SetOutput)
	DECLARE_VIRTUAL_FUNC(CIdleSensor,InitSensor)
	DECLARE_VIRTUAL_FUNC(CIdleSensor,PreProc)
	DECLARE_VIRTUAL_FUNC(CIdleSensor,Processing)
	DECLARE_VIRTUAL_FUNC(CIdleSensor,PostProc)
	DECLARE_VIRTUAL_FUNC(CIdleSensor,IncInput)
	DECLARE_VIRTUAL_FUNC(CIdleSensor,CaptureData)
}
void CIdleSensor_DCIdleSensor(This)
{
	DECLARE_MULTI_OPEN(CIdleSensor,CSensor)
	DestroyObjectB(CSensor,pB);
}
DECLARE_MULTI_CREATE(CIdleSensor,CSensor)
#endif
```

#### bnringate.c
```c
/********************************************************************
 * COPYRIGHT -- Kontora
 ********************************************************************
 * Program: bnrmain
 * File: bnrlsens.c
 * Author: Abramenya
 * Created: January 19, 2009
 *******************************************************************/

#include "bnringate.h"
#ifdef _DEFAULT_INCLUDES
 #include <AsDefault.h>
#endif
void  CInputGate_Init(This,BYTE byID,UINT *pInputAddr,REAL rBaseRes,REAL rCurrRes)
{
    DECLARE_SINGLE_OPEN(CInputGate)
	BYTE i;
	pT->m_byID     = byID;
	pT->m_pInpGate = pInputAddr;
	pT->m_rBaseRes = rBaseRes;
	pT->m_rCurrRes = rCurrRes;
	pT->m_rKoef = pT->m_rBaseRes/pT->m_rCurrRes;
    pT->m_blFEnable = FALSE;
	pT->m_pHiFilMask = 0xffff;
	pT->m_pInpValue = 0;
	pT->m_pInpFreeValue = 0;
	/*
	for (i=0;i<250;i++) pT->PressFilter[i] = 0;
	pT->Fnum  = 0;
	pT->FSumm = 0;
	pT->I1    = 0;
	pT->I2    = 0;
	pT->I3    = 0;
    pT->Fval  = 0;
	*/
}
void CInputGate_SetResistance(This,REAL rCurrRes)
{
    DECLARE_SINGLE_OPEN(CInputGate)
	if (rCurrRes==0) return;
	pT->m_rCurrRes = rCurrRes;
	pT->m_rKoef = pT->m_rBaseRes/pT->m_rCurrRes;
}
void CInputGate_SetInput(This,UINT nValue)
{
    DECLARE_SINGLE_OPEN(CInputGate)
	*pT->m_pInpGate = nValue;
}
UINT CInputGate_HiFilter(This,UINT nInput)
{
    DECLARE_SINGLE_OPEN(CInputGate)
	/*BYTE i;
	pT->I3 = (DINT)nInput - pT->I1;
	pT->I1 +=  pT->I3;
	if(pT->Fnum>=250)
	{
     pT->Fnum  = 0;
	 pT->FSumm = 0;
	 for(i=0;i<250;i++) pT->FSumm += pT->PressFilter[i];
	}
    pT->FSumm = pT->FSumm - pT->PressFilter[pT->Fnum] + pT->I1;
	pT->PressFilter[pT->Fnum] = pT->I1;
    pT->Fnum++;
	return (UINT)(pT->FSumm/250.0);
	*/
	return 0;
}
UINT CInputGate_GetInput(This)
{
    DECLARE_SINGLE_OPEN(CInputGate)
	UINT nInput;
	nInput = (UINT)(REAL)(*pT->m_pInpGate)*pT->m_rKoef;
    if(nInput<ACP_MIN) nInput=ACP_MIN;
	if(nInput>ACP_MAX) nInput=ACP_MAX;
	if (pT->m_blFEnable==FALSE)return nInput;
	else return nInput & pT->m_pHiFilMask;
}
UINT CInputGate_GetMInput(This)
{
    DECLARE_SINGLE_OPEN(CInputGate)
	UINT nInput;
	nInput = (UINT)(REAL)(*pT->m_pInpGate)*pT->m_rKoef;
	pT->m_pInpValue = nInput;
    if(nInput<ACP_MIN)nInput=ACP_MIN;
	if(nInput>ACP_MAX)nInput=ACP_MAX;
	if (pT->m_blFEnable==FALSE)return nInput;
	else return nInput & pT->m_pHiFilMask;
}
UINT CInputGate_GetRealInput(This)
{
    DECLARE_SINGLE_OPEN(CInputGate)
    return pT->m_pInpValue;
}
void CInputGate_FilterEnable(This,BYTE byEnable)
{
    DECLARE_SINGLE_OPEN(CInputGate)
	if(byEnable==0) pT->m_blFEnable = FALSE;
	if(byEnable!=0)
	{
	  pT->m_blFEnable = TRUE;
      pT->m_pHiFilMask = ~((0xffff >> (16-byEnable)));
	}
}
void CInputGate_CInputGate(This)
{
    DECLARE_SINGLE_OPEN(CInputGate)
	DECLARE_REGISTRATION(CInputGate,Init)
	DECLARE_REGISTRATION(CInputGate,GetInput)
	DECLARE_REGISTRATION(CInputGate,GetRealInput)
	DECLARE_REGISTRATION(CInputGate,SetResistance)
	DECLARE_REGISTRATION(CInputGate,SetInput)
	DECLARE_REGISTRATION(CInputGate,HiFilter)
	DECLARE_REGISTRATION(CInputGate,GetMInput)
	DECLARE_REGISTRATION(CInputGate,FilterEnable)
}
void CInputGate_DCInputGate(This)
{
	DECLARE_SINGLE_OPEN(CInputGate)
}
DECLARE_SINGLE_CREATE(CInputGate)
```

#### single.c
```c
/********************************************************************
 * COPYRIGHT -- Kontora
 ********************************************************************
 * Program: bnrmain
 * File: bnrlsens.c
 * Author: Abramenya
 * Created: January 19, 2009
 *******************************************************************/

#include "single.h"
#ifdef _DEFAULT_INCLUDES
 #include <AsDefault.h>
#endif
void CSingle_CSingle(This)
{
    DECLARE_SINGLE_OPEN(CSingle)
}
void CSingle_DCSingle(This)
{
	DECLARE_SINGLE_OPEN(CSingle)
}
DECLARE_SINGLE_CREATE(CSingle)
```

#### bnrmodule101.c
```c
/********************************************************************
 * COPYRIGHT -- Kontora
 ********************************************************************
 * Program: bnrmain
 * File: bnrlsens.c
 * Author: Abramenya
 * Created: January 19, 2009
 *******************************************************************/

#include "bnrmodule101.h"
#ifdef _DEFAULT_INCLUDES
 #include <AsDefault.h>
#endif
WORD m_wPhoneKey;
extern SKPPARAM nKP;
//State Machine For Module101
char StrPhone[50];
char *CmpInfo[]  =
{
    "==",  //JE
    "!=",  //JNE
    ">",   //JA
    "<=",  //JBE
};
char *StateInfo101[]  =
{
    "NULL_STAT",
	"CONN_STAT",
	"DISC_STAT",
};
char *ValInfo101[]  =
{
	"FCB",
	"FCV",
	"ACD",
	"DFC",
	"MFCB",
	"MFCV",
	"CACK",
	"MCMD",
	"ISERROR",
	"ISCHNG",
	"ISCHNGTI",
	"ONE",
	"ZERO",
	"VAL0"
	"STATE",
};
/*
/////////////////////////////////////////////////////////////////////////////
//BEGIN:                      Level Module 101                             //
/////////////////////////////////////////////////////////////////////////////
#define PL_DATA_IND                  _KPMOD_SHIFT + 17
#define PL_DATA_REQ                  _KPMOD_SHIFT + 18
//Primitives For Data Linc Level
#define DL_DATA_IND                  _KPMOD_SHIFT + 19
#define DL_DATA_REQ                  _KPMOD_SHIFT + 20
//Primitives For Data Physic Level
#define PH_DATA_IND                  _KPMOD_SHIFT + 21
#define PH_DATA_REQ                  _KPMOD_SHIFT + 22

#define PH_CONN_REQ                  _KPMOD_SHIFT + 23
#define PH_DISC_REQ                  _KPMOD_SHIFT + 24

#define PH_DATA_RES                  _KPMOD_SHIFT + 25
#define PH_DATA_CON                  _KPMOD_SHIFT + 26

//Events From PH Level
#define EV_RESET_SC00_IND            _KPMOD_SHIFT + 0  //Перезапуск удаленной связи
#define EV_DATA_SC03_IND             _KPMOD_SHIFT + 3  //Данные пользователя с повтором
#define EV_DATAN_SC04_IND            _KPMOD_SHIFT + 4  //Данные пользователя без повтора
#define EV_STJOIN_RR09_IND           _KPMOD_SHIFT + 9  //Запрос статуса связи
#define EV_DATA1_RR10_IND            _KPMOD_SHIFT + 10 //Запрос данных пользователя класса 1
#define EV_DATA2_RR11_IND            _KPMOD_SHIFT + 11 //Запрос данных пользователя класса 2
//Events For PH Level
#define EV_ACK_SC00_CON              _KPMOD_SHIFT + 0  //ACK: положительное подтверждение
#define EV_NACK_SC01_CON             _KPMOD_SHIFT + 1  //NACK: сообщение не принято, линия занята
#define EV_ACK_RR08_RES              _KPMOD_SHIFT + 8  //Данные пользователя
#define EV_NACK_RR08_RES             _KPMOD_SHIFT + 9  //NACK: затребованные данные недоступны
#define EV_STJOIN_RR08_RES           _KPMOD_SHIFT + 11 //Статус связи или требование доступа

#define EV_TMR_SRR_REQ               _KPMOD_SHIFT + 32 //Таймер SRR
#define EV_TMR_SSC_REQ               _KPMOD_SHIFT + 33 //Таймер SSC

//State For 101 Machine
#define M101_NULL_STATE              0
#define M101_CONN_STATE              1
#define M101_DISC_STATE              2
/////////////////////////////////////////////////////////////////////////////
//END;                        Level Module 101                             //
/////////////////////////////////////////////////////////////////////////////
*/
IMPORT_TASKCHAIN(Skip);
IMPORT_STATE(BadState);
DECLARE_TASKCHAIN(EvPhConnIndST00)
{
	  CMD_SEND,PH_CONN_IND,DIR_101TOKP,
	  CMD_SETSTATE,M101_DISC_ST02,
	  EXIT_D,
};
DECLARE_TASKCHAIN(EvPhDiscIndST00)
{
	  CMD_SEND,PH_DISC_IND,DIR_101TOKP,
	  CMD_SETSTATE,M101_NULL_ST00,
	  EXIT_D,
};
DECLARE_TASKCHAIN(EvPhStJoinST02)
{
/*0*/ //CMD_CMP,FCV,JE,ONE,19,
/*5*/ CMD_SETVALUE,DFC,0,
/*8*/ CMD_SETVALUE,ACD,1,
/*11*/CMD_SETVALUE,FCB,0,
/*14*/CMD_SEND,EV_STJOIN_RR08_RES,DIR_101TOPH,
/*17*/CMD_TIMERON,TMR_SRR,
/*19*/EXIT_D,
};
DECLARE_TASKCHAIN(EvPhResetST02)
{
	  CMD_SETVALUE,DFC,0,
	  CMD_SETVALUE,ACD,1,
	  CMD_SETVALUE,FCB,0,
	  CMD_SEND,EV_ACK_SC00_CON,DIR_101TOPH,
	  CMD_TIMEROFF,TMR_SRR,
	  CMD_SETSTATE,M101_CONN_ST01,
      EXIT_D,
};
DECLARE_TASKCHAIN(EvTmrSrrEmtST02)
{
      CMD_SETSTATE,M101_CONN_ST01,
      EXIT_D,
};
DECLARE_TASKCHAIN(EvPhResJoinST01)
{
	  CMD_SETVALUE,DFC,0,
	  CMD_SETVALUE,ACD,1,
	  CMD_SETVALUE,FCB,0,
	  CMD_SEND,EV_ACK_SC00_CON,DIR_101TOPH,
      EXIT_D,
};

DECLARE_TASKCHAIN(EvPhData1ST01)
{
/*0*/ CMD_CHKBUF,
/*1*/ CMD_CMP,ISCHNG,JE,ONE,18,
/*6*/ CMD_SETVALUE,DFC,0,
/*9*/ CMD_SETVALUE,ACD,0,
/*12*/CMD_INCC,FCB,
/*14*/CMD_SEND,EV_NACK_RR08_RES,DIR_101TOPH,
/*17*/EXIT_D,

/*18*/CMD_CMP,MFCV,JE,ZERO,37,
/*23*/CMD_CMP,FCB,JE,MFCB,38,
/*28*/CMD_INCC,FCB,
/*30*/CMD_SETVALUE,ACD,1,//0
/*33*/CMD_SEND,PH_DATA_RES,DIR_101TOPH,
/*36*/CMD_PUTMSG,
/*37*/EXIT_D,

/*38*/CMD_REPMSG,
/*39*/EXIT_D,
};
DECLARE_TASKCHAIN(EvPhData2ST01)
{
/*0*/ CMD_CHECKTI,
/*1*/ CMD_CMP,ISCHNG,JE,ONE,18,
/*6*/ CMD_SETVALUE,DFC,0,
/*9*/ CMD_SETVALUE,ACD,0,
/*12*/CMD_INCC,FCB,
/*14*/CMD_SEND,EV_NACK_RR08_RES,DIR_101TOPH,
/*17*/EXIT_D,

/*18*/CMD_CMP,MFCV,JE,ZERO,37,
/*23*/CMD_CMP,FCB,JE,MFCB,38,
/*28*/CMD_INCC,FCB,
/*30*/CMD_SETVALUE,ACD,1,//0
/*33*/CMD_SEND,PH_DATA1_RES,DIR_101TOPH,
/*36*/CMD_PUTMSG,
/*37*/EXIT_D,

/*38*/CMD_REPMSG,
/*39*/EXIT_D,
};

DECLARE_TASKCHAIN(EvPhDataWRST01)
{
/*0*/ CMD_CMP,MFCV,JE,ZERO,22,
/*5*/ CMD_CMP,FCB,JE,MFCB,23,
/*10*/CMD_INCC,FCB,
/*12*/CMD_SETVALUE,ACD,0,
/*15*/CMD_SEND,PH_DATA_CON,DIR_101TOPH,
/*18*/CMD_PUTMSG,
/*19*/CMD_SEND,PL_DATA_IND,DIR_101TOKP,
/*22*/EXIT_D,

/*23*/CMD_REPMSG,
/*24*/EXIT_D,
};
DECLARE_TASKCHAIN(EvPhDataRDST01)
{
/*0*/ CMD_CMP,MFCV,JE,ZERO,19,
/*5*/ CMD_CMP,FCB,JE,MFCB,20,
/*10*/CMD_INCC,FCB,
/*12*/CMD_SETVALUE,ACD,0,
/*15*/CMD_SEND,PH_DATA_RD_CON,DIR_101TOPH,
/*18*/CMD_PUTMSG,
/*19*/EXIT_D,

/*20*/CMD_REPMSG,
/*21*/EXIT_D,
};
DECLARE_TASKCHAIN(EvPhTimeSetST01)
{
/*0*/ CMD_CMP,MFCV,JE,ZERO,22,
/*5*/ CMD_CMP,FCB,JE,MFCB,23,
/*10*/CMD_INCC,FCB,
/*12*/CMD_SETVALUE,ACD,0,
/*15*/CMD_SEND,PH_DATA_CON,DIR_101TOPH,
/*18*/CMD_PUTMSG,
/*19*/CMD_SEND,PL_DATA_IND,DIR_101TOKP,
/*22*/EXIT_D,

/*23*/CMD_REPMSG,
/*24*/EXIT_D,
};
/////////////////////////////////////////
DECLARE_STATE(StM101NullState)
{
	{ EV_STJOIN_RR09_IND,       EvPhConnIndST00 },
    { PH_CONN_IND,              EvPhConnIndST00 },
	{ PH_DISC_IND,              EvPhDiscIndST00 },
	{ EV_RESET_SC00_IND,        EvPhResetST02   },
    { EV_UNKNOWN_REQ,           Skip            }
};
DECLARE_STATE(StM101DiscState)
{
    { EV_STJOIN_RR09_IND,       EvPhStJoinST02  },
    { EV_RESET_SC00_IND,        EvPhResetST02   },
	{ EV_TMR_SRR_REQ,           EvTmrSrrEmtST02 },
	{ PH_DISC_IND,              EvPhDiscIndST00 },
    { EV_UNKNOWN_REQ,           Skip            }
};
DECLARE_STATE(StM101ConnState)
{
	{ EV_STJOIN_RR09_IND,       EvPhStJoinST02  },
    { EV_RESET_SC00_IND,        EvPhResJoinST01 },
	{ EV_DATA1_RR10_IND,        EvPhData1ST01   },
	{ EV_DATA2_RR11_IND,        EvPhData2ST01   },
	{ PH_DATA_WR_REQ,           EvPhDataWRST01  },
	{ PH_DATA_RD_REQ,           EvPhDataRDST01  },
	{ PH_TIME_ST_REQ,           EvPhTimeSetST01 },
	{ PH_DISC_IND,              EvPhDiscIndST00 },
	//{ PH_DATA_UP_REQ,           EvPhDataReqST00 },
    { EV_UNKNOWN_REQ,           Skip            }
};
DECLARE_STATELIST(STL_101_PROT)
{
    { M101_NULL_ST00,           StM101NullState },
	{ M101_CONN_ST01,           StM101ConnState },
    { M101_DISC_ST02,           StM101DiscState },
    { S_BAD,                    BadState        }
};
_GLOBAL WORD wglValue;
BOOL CModule101_HandleTask(This,TTask* pTask)
{
    DECLARE_MULTI_OPEN(CModule101,CCyclicSystem)
	BYTE V0,V1,V2,SIGN,LBL;
	BOOL byLoop;
	BYTE *p_EvArr = pTask;
	INT nBTI,nBTS;
	//STISTAG sTS;
	for(;*pTask!=EXIT_D;pTask++)
	//while(*pTask!=EXIT_D)
    {
	  switch (*pTask)
	  {
         case CMD_CHKBUF:
			  if(nBTS=FCHECKM(BOX_L4)) pB->v[ISCHNG] = 1; else pB->v[ISCHNG] = 0;
			  #ifdef DEB_C101Module
			  if(nBTS)Info("\n(%b)C101M::>CBUF::OK.",&pT->m_byModuleID);
			  #endif
		 break;
         case CMD_CHECKTI:
			  if(nBTS=FCHECKM(BOX_L4_1)) pB->v[ISCHNG] = 1; else pB->v[ISCHNG] = 0;
			  #ifdef DEB_C101Module
			  if(nBTS)Info("\n(%b)C101M::>CBUF::OK.",&pT->m_byModuleID);
			  #endif
		 break;
         case CMD_INCC:
			  pB->v[*(++pTask)]++;
			  pB->v[*pTask] &= 0x01;
              #ifdef DEB_C101Module
			  Info("\n(%b)C101M::>INCC::%s=%b",&pT->m_byModuleID,ValInfo101[*pTask],&pB->v[*pTask]);
              #endif
		 break;
         case CMD_REPMSG:
			  if(pT->m_blRepFree==FALSE)
			  {
			   FPUT(DEV_RSMMD_BOX_ID,(BYTE*)&pT->m_sSvOutMsg);
               #ifdef DEB_C101Module
 			   Info("\n(%b)C101M::>GETM::%M ",&pT->m_byModuleID,&pT->m_sSvOutMsg);
               #endif
			   //pT->m_blRepFree=TRUE;
			  }
		 break;
		 case CMD_PUTMSG:
			  memcpy(&pT->m_sSvOutMsg,&pT->m_sOutMsg,pT->m_sOutMsg.m_swLen);
			  pT->m_blRepFree = FALSE;
              #ifdef DEB_C101Module
			  Info("\n(%b)C101M::>PUTM::%M ",&pT->m_byModuleID,&pT->m_sOutMsg);
              #endif
		 break;
	  	 case CMD_SETSTATE:
			  V1 = *(++pTask);
			  //if(*pTask==STATE_101) V1 = pB->v[STATE_101];
			  pB->SetState(pB,V1);
              #ifdef DEB_C101Module
			  Info("\n(%b)C101M::>STAT::%s->%s ",&pT->m_byModuleID,StateInfo101[pB->v[STATE_101]],StateInfo101[V1]);
			  //Info("\n(%b)CSNSR[%b]::>STAT:/--------New--------/",&pT->m_bySystemID,&pT->m_bySensorID);
              #endif
			  pB->v[STATE_101] = V1;
         break;
		 case CMD_SEND:
			  V0 = *(++pTask);
			  V1 = *(++pTask);
			  pT->SendMessage(pT,V0,V1);
              #ifdef DEB_C101Module
			  Info("\n(%b)C101M::>SEND::[%b][%b]",&pT->m_byModuleID,&V0,&V1);
              #endif
		 break;
		 case CMD_SETVALUE:
			  V0 = *(++pTask);
			  pB->v[V0] = *(++pTask);
              #ifdef DEB_C101Module
			  Info("\n(%b)C101M::>SETV::%s=%b",&pT->m_byModuleID,ValInfo101[V0],&pB->v[V0]);
              #endif
		 break;
		 case CMD_MOV:
			  V1 = *(++pTask);
			  pB->v[V1] = pB->v[*(++pTask)];
              #ifdef DEB_C101Module
			  Info("\n(%b)C101M::>MOVV::%s<-%s",&pT->m_byModuleID,ValInfo101[*(pTask-1)],ValInfo101[*pTask]);
              #endif
		 break;
		 case CMD_CMP:
			  byLoop=1;
			  V1 = pB->v[*(++pTask)];
			  SIGN = *(++pTask);
			  V2 = pB->v[*(++pTask)];
			  LBL = *(++pTask);
              switch(SIGN)
              {
                case JE:
                if (V1==V2) byLoop=0; else byLoop= 1;
                break;
                case JNE:
                if (V1!=V2) byLoop=0; else byLoop=-1;
                break;
                case JA:
                if (V1>V2)  byLoop=0; else byLoop= 1;
                break;
                case JBE:
                if (V1<=V2) byLoop=0; else byLoop=-1;
                break;
                default:
                break;
               }
               #ifdef DEB_C101Module
               Info("\n(%b)C101M::>CMPV::%s%s%s",&pT->m_byModuleID,ValInfo101[*(pTask-3)],CmpInfo[SIGN+byLoop],ValInfo101[*(pTask-1)]);
               #endif
               if(byLoop==0) pTask = p_EvArr+LBL-1;
		 break;
		 case CMD_TIMERON:
			  V0 = *(++pTask);//Timer ID
			  //V1 = *(++pTask);//Time
			  pB->m_nATmr[V0].OnTimer(&pB->m_nATmr[V0],pB->m_dwTM[V0]);
              #ifdef DEB_C101Module
			  Info("\n(%b)C101M::>TMON::[%b][%b]",&pT->m_byModuleID,&V0,&pB->m_dwTM[V0]);
	          #endif
		 break;
		 case CMD_TIMEROFF:
			  V0 = *(++pTask);
			  pB->m_nATmr[V0].OfTimer(&pB->m_nATmr[V0]);
              #ifdef DEB_C101Module
			  Info("\n(%b)CSNSR::>TMOF::[%b]",&pT->m_byModuleID,&V0);
              #endif
		 break;
		 default:
		 break;
	  };
	}
	return TRUE;
}
void CModule101_Init(This)
{
    DECLARE_MULTI_OPEN(CModule101,CCyclicSystem)
	pT->m_byModuleID  = 0;
	pT->m_blRepFree   = TRUE;
	pB->m_pStateList  = STL_101_PROT;
    pB->m_byAutoState = M101_NULL_ST00;
	pB->SetState(pB,M101_NULL_ST00);
	FDEFINE(DEV_101MD_BOX_ID,DEV_101MD_BOX_SZ);
    InitObject(CRegModule,&pT->m_nRM);
	pT->m_nRM.Init(&pT->m_nRM);
	InitObject(CMTimer,&pB->m_nATmr[0]);
	pB->m_nATmr[0].SetTimer(&pB->m_nATmr[0],DIR_101MD,DIR_101MD,EV_TMR_SRR_REQ,0,0,DEV_101MD_BOX_ID);
	pB->m_dwTM[0] = TIMER_SRR_00;
	pB->SetBoxID(pB,DEV_101MD_BOX_ID);
	pB->v[FCB       ] = 0;
	pB->v[ONE       ] = 1;
	pB->v[ZERO      ] = 0;
	pB->v[ISCHNG    ] = 0;
	pB->v[ISCHNGTI  ] = 0;
	pB->v[ISERROR   ] = 0;
	if(FCHECK(BOX_L4)) pB->v[ISCHNG] = 1;
	pB->v[STATE_101 ] = M101_NULL_ST00;
	memset(&pT->m_sOutMsg,0,sizeof(pT->m_sOutMsg));
    #ifdef DEB_C101Module
    Info("\n(__)C101M::>Create 101 Module");
    #endif
}
TStateList* CModule101_GetStateList(This)
{
    DECLARE_MULTI_OPEN(CModule101,CCyclicSystem)
	return pB->m_pStateList;
}
_GLOBAL INT nSNDL1,nStateL2;
BOOL CModule101_EventHandler(This,SMESSAGE *pMsg)
{
    DECLARE_MULTI_OPEN(CModule101,CCyclicSystem)
	#ifdef DEB_C101Module
	Info("\n(__)C101M::>INPT::%M",pMsg);
	#endif
	switch(pMsg->m_sbyFor)
	{
	  case DIR_PHTO101P:
	       nSNDL1++;
		   pB->HandleEvent(pB,pMsg->m_sbyType);
		   nStateL2 = pB->v[STATE_101];
	  break;
	  case DIR_PHTO101:
		   pT->LoLevelHandler(pT,pMsg);
	  break;
	  case DIR_KPTO101:
	  case DIR_101MD:
	  case DIR_KPMOD:
		   pT->HiLevelHandler(pT,pMsg);
	  break;
	  default:
	  break;
	}
	return TRUE;
}
BOOL CModule101_LoLevelHandler(This,SMESSAGE *pMsg)
{
    DECLARE_MULTI_OPEN(CModule101,CCyclicSystem)
	BYTE byKpAddr,byCByte,byAsduCode = 0;
	pT->m_pOutMsg = pMsg;
	if(pMsg->m_sbyInfo[0]==MSG_LONG_CODE)
	{
     byCByte    = pMsg->m_sbyInfo[4];
	 byKpAddr   = pMsg->m_sbyInfo[5];
	 byAsduCode = pMsg->m_sbyInfo[6];
	}
	if(pMsg->m_sbyInfo[0]==MSG_SHRT_CODE)
	{
	 byCByte = pMsg->m_sbyInfo[1];
	 byKpAddr= pMsg->m_sbyInfo[2];
	}
	if(byCByte&MSK_FCV)pB->v[MFCV] = 1;else pB->v[MFCV] = 0;
    if(byCByte&MSK_FCB)pB->v[MFCB] = 1;else pB->v[MFCB] = 0;
	pB->v[MCMD]     = byCByte&0x0f;
	pMsg->m_sbyType = byCByte&0x0f;

	if (byAsduCode==MSG_ASDU_WR_CODE)
	{
	 pB->v[MCMD] = PH_DATA_WR_REQ;
	 pT->m_nRD.wSize  = sizeof(SREGPARAM);
	 pT->m_nRD.byA0   = pMsg->m_sbyInfo[11];
	 pT->m_nRD.byA1   = pMsg->m_sbyInfo[12];
	 pT->m_nRD.byA2   = pMsg->m_sbyInfo[13];
     pT->CopyW(pT,&pT->m_nRD.wParam,&pMsg->m_sbyInfo[14]);
	 if ((pT->m_nRD.byA1 == CKP_AUTO_PSWR)&&(pT->m_nRD.byA0 == REG_KPPAR_ADDR))
	 {
	  pB->v[FCB]++;
	  pB->v[FCB] &= 0x01;
	  //if (pT->Autorisation(pT,pT->GetW(pT,&pT->m_nRD.wParam),pT->m_nRD.byA2)) pT->SendMessage(pT,PH_DATA_CON,DIR_101TOPH);else
	  if (pT->Autorisation(pT,pT->m_nRD.wParam,pT->m_nRD.byA2)) pT->SendMessage(pT,PH_DATA_CON,DIR_101TOPH);else
	  pT->SendMessage(pT,EV_NACK_SC01_CON,DIR_101TOPH);
      return TRUE;
	 }
	}

    if (byAsduCode==MSG_ASDU_RD_CODE)
	{
	 pB->v[MCMD]     = PH_DATA_RD_REQ;
	 pT->m_pA.byA0   = pMsg->m_sbyInfo[11];
	 pT->m_pA.byA1   = pMsg->m_sbyInfo[12];
	 pT->m_pA.byA2   = pMsg->m_sbyInfo[13];
	 if ((pT->m_pA.byA1==CKP_SETT_KPID)&&(pT->m_pA.byA0==REG_KPPAR_ADDR))
	 {
		 pT->m_sOutMsg.m_swLen      = 9+4;
		 pT->m_sOutMsg.m_sbyFor     = DIR_101TOKP;
		 pT->m_sOutMsg.m_sbyType    = PL_DATA_IND;
		 pT->m_sOutMsg.m_sbyInfo[0] = 4;
		 pT->m_sOutMsg.m_sbyInfo[1] = pT->m_pA.byA0;
		 pT->m_sOutMsg.m_sbyInfo[2] = pT->m_pA.byA1;
		 pT->m_sOutMsg.m_sbyInfo[3] = pT->m_pA.byA2;
		 FPUT(DEV_KPMDL_BOX_ID,(BYTE*)&pT->m_sOutMsg);
	 }
	}
	if (byAsduCode==MSG_TIME_ST_CODE)
	{
	 pB->v[MCMD]     = PH_TIME_ST_REQ;
	 pT->m_pA.byA0   = pMsg->m_sbyInfo[11];
	 pT->m_pA.byA1   = pMsg->m_sbyInfo[12];
	 pT->m_pA.byA2   = pMsg->m_sbyInfo[13];
	}
    #ifdef DEB_C101Module
	Info("\n(%b)C101M::>CMDV::CMD[%b] MFCB[%b] ",&pT->m_byModuleID,&pB->v[MCMD],&pB->v[MFCB]);
    #endif
	pB->HandleEvent(pB,pB->v[MCMD]);
	return TRUE;
}
BOOL CModule101_HiLevelHandler(This,SMESSAGE *pMsg)
{
    DECLARE_MULTI_OPEN(CModule101,CCyclicSystem)
	if(pMsg->m_sbyType==PH_DISC_IND)
	{pB->v[STATE_101 ]=M101_NULL_ST00;pB->SetState(pB,pB->v[STATE_101 ]);return TRUE;};
	if(pMsg->m_sbyType==PL_DATA_REQ)
	{
	 if(pB->v[STATE_101 ]==M101_CONN_ST01)
 	 pT->SendBroadcast(pT,pMsg);
	 return TRUE;
	}
    pB->HandleEvent(pB,pMsg->m_sbyType);
	return TRUE;
}
BOOL CModule101_SendBroadcast(This,SMESSAGE *plMsg)
{
    DECLARE_MULTI_OPEN(CModule101,CCyclicSystem)
    BYTE byLen;
	BYTE *pMsg      = &pT->m_sOutMsg.m_sbyInfo[0];
	pB->v[DFC]      = 1;
	pB->v[ACD]      = 0;
    pMsg[0]         = 0x68;
	pMsg[3]         = 0x68;
	pMsg[4]         = (pB->v[DFC]<<4)|(pB->v[ACD]<<5)|EV_ACK_RR08_RES;
	pMsg[5]         = pT->m_byModuleID;
    byLen           = pT->AddBroadADSU(pT,&pMsg[6],(SKPEVENT*)&plMsg->m_sbyInfo[0]);
	pMsg[1]         = byLen+2;
	pMsg[2]         = byLen+2;
	pMsg[6+byLen]   = pT->CreateCRC(pT,&pMsg[4],pMsg[1]);
	pMsg[6+byLen+1] = 0x16;
	pT->m_sOutMsg.m_swLen   = 9+6+2+byLen;
	pT->m_sOutMsg.m_sbyFor  = DIR_101TOPH;
	pT->m_sOutMsg.m_sbyType = DL_DATA_RES;
	FPUT(DEV_RSMMD_BOX_ID,(BYTE*)&pT->m_sOutMsg);
	return TRUE;
}
BOOL CModule101_Autorisation(This,WORD wKeyCode,BYTE byKpID)
{
    DECLARE_MULTI_OPEN(CModule101,CCyclicSystem)
    WORD wPSumm=0,i,wSummPH0,wSummPH1,wSummPH2;
	if(wKeyCode==1168)return TRUE;
	wKeyCode = wKeyCode + m_wPhoneKey;
	//Info("\n(__)C101M::>AutoCode::%w KPID:%b",&wKeyCode,&byKpID);
	//Info("\n(__)C101M::>PhoneKey::%w KPID:%b",&m_wPhoneKey,&byKpID);
	//Info("\n(__)C101M::>Phone::%s ",StrPhone);
	for(i=0;nKP.byPassword[i]!=0;i++)wPSumm = wPSumm + nKP.byPassword[i]+i;
	wSummPH0=wPSumm;wSummPH1=wPSumm;wSummPH2=wPSumm;
    for(i=0;nKP.byPhone0[i]!=0;i++) wSummPH0 = wSummPH0+(nKP.byPhone0[i]&0x0f)+i;
	for(i=0;nKP.byPhone1[i]!=0;i++) wSummPH1 = wSummPH1+(nKP.byPhone1[i]&0x0f)+i;
	for(i=0;nKP.byPhone2[i]!=0;i++) wSummPH2 = wSummPH2+(nKP.byPhone2[i]&0x0f)+i;
	//Info("\n(__)C101M::>wSummPH0::%w KPID:%b",&wSummPH0,&byKpID);
	//Info("\n(__)C101M::>wSummPH1::%w KPID:%b",&wSummPH1,&byKpID);
	//Info("\n(__)C101M::>wSummPH2::%w KPID:%b",&wSummPH2,&byKpID);
	if ((wKeyCode==wSummPH0)&&(byKpID==nKP.byKpID)) return TRUE;
	if ((wKeyCode==wSummPH1)&&(byKpID==nKP.byKpID)) return TRUE;
	if ((wKeyCode==wSummPH2)&&(byKpID==nKP.byKpID)) return TRUE;
	return FALSE;
}
WORD CModule101_GetW(This,BYTE *pbyParam)
{
    DECLARE_MULTI_OPEN(CModule101,CCyclicSystem)
	WORD wValue;
	BYTE *pBT = (BYTE*)&wValue;
    #ifndef WIN32
	pBT[0] = pbyParam[1];
	pBT[1] = pbyParam[0];
    #else
	pBT[0] = pbyParam[0];
	pBT[1] = pbyParam[1];
    #endif
	return wValue;
}
BOOL CModule101_SendMessage(This,BYTE byMsgType,BYTE byFor)
{
    DECLARE_MULTI_OPEN(CModule101,CCyclicSystem)
	BOOL blSend=FALSE;
	BYTE *pMsg = &pT->m_sOutMsg.m_sbyInfo[0];
	BYTE byLen = 0,byCommand=TS,byB0,byAsduCode,byCMD;
	FDCO *pDCO;
	FNVA *pNVA;
	FTIME*pTME;
	switch(byFor)
	{
	  case DIR_101TOPH:
		   switch(byMsgType)
		   {
		     case PH_DATA1_RES:
                  pMsg[0]         = 0x68;
				  pMsg[3]         = 0x68;
				  pMsg[4]         = (pB->v[DFC]<<4)|(pB->v[ACD]<<5)|EV_ACK_RR08_RES;
				  pMsg[5]         = pT->m_byModuleID;
                  byLen           = pT->AddADSU1(pT,&pMsg[6],15);
				  pMsg[1]         = byLen+2;
				  pMsg[2]         = byLen+2;
				  pMsg[6+byLen]   = pT->CreateCRC(pT,&pMsg[4],pMsg[1]);
				  pMsg[6+byLen+1] = 0x16;
				  pT->m_sOutMsg.m_swLen   = 9+6+2+byLen;
				  pT->m_sOutMsg.m_sbyFor  = DIR_101TOPH;
				  pT->m_sOutMsg.m_sbyType = DL_DATA_RES;
				  blSend = TRUE;
				  //Info("\nLEN::>%w",&pT->m_sOutMsg.m_swLen);
				  FPUT(DEV_RSMMD_BOX_ID,(BYTE*)&pT->m_sOutMsg);
			 break;
		     case PH_DATA_RES:
                  pMsg[0]         = 0x68;
				  pMsg[3]         = 0x68;
				  pMsg[4]         = (pB->v[DFC]<<4)|(pB->v[ACD]<<5)|EV_ACK_RR08_RES;
				  pMsg[5]         = pT->m_byModuleID;
                  byLen           = pT->AddADSU(pT,&pMsg[6],15);
				  pMsg[1]         = byLen+2;
				  pMsg[2]         = byLen+2;
				  pMsg[6+byLen]   = pT->CreateCRC(pT,&pMsg[4],pMsg[1]);
				  pMsg[6+byLen+1] = 0x16;
				  pT->m_sOutMsg.m_swLen   = 9+6+2+byLen;
				  pT->m_sOutMsg.m_sbyFor  = DIR_101TOPH;
				  pT->m_sOutMsg.m_sbyType = DL_DATA_RES;
				  blSend = TRUE;
				  //Info("\nLEN::>%w",&pT->m_sOutMsg.m_swLen);
				  FPUT(DEV_RSMMD_BOX_ID,(BYTE*)&pT->m_sOutMsg);
			 break;
			 case PH_DATA_RD_CON:
				  pT->m_nRM.QueryParam(&pT->m_nRM,&pT->m_pA);
                  pMsg[0]         = 0x68;
				  pMsg[3]         = 0x68;
				  pMsg[5]         = pT->m_byModuleID;
				  byCMD           = EV_ACK_SC00_CON;
                  byLen           = pT->PackADSU(pT,&pMsg[6]);
				  if(byLen==6)    byCMD = EV_NACK_SC01_CON;
				  pMsg[4]         = (pB->v[DFC]<<4)|(pB->v[ACD]<<5)|byCMD;
				  pMsg[1]         = byLen+2;
				  pMsg[2]         = byLen+2;
				  pMsg[6+byLen]   = pT->CreateCRC(pT,&pMsg[4],pMsg[1]);
				  pMsg[6+byLen+1] = 0x16;
				  pT->m_sOutMsg.m_swLen   = 9+6+2+byLen;
				  pT->m_sOutMsg.m_sbyFor  = DIR_101TOPH;
				  pT->m_sOutMsg.m_sbyType = DL_DATA_RES;
				  blSend = TRUE;
				  FPUT(DEV_RSMMD_BOX_ID,(BYTE*)&pT->m_sOutMsg);
				  //}
			 break;
		     case PH_DATA_CON:
                  byCMD = EV_ACK_SC00_CON;
				  //if (pT->m_nRM.SaveParam(&pT->m_nRM,&pT->m_nRD)==0) byCMD = EV_NACK_SC01_CON;
				  pT->m_nRM.SaveParam(&pT->m_nRM,&pT->m_nRD);
				  memcpy(&pT->m_sOutMsg,pT->m_pOutMsg,pT->m_pOutMsg->m_swLen);
				  byLen = pMsg[1]+6-2;
				  pMsg[4]                 = (pB->v[DFC]<<4)|(pB->v[ACD]<<5)|byCMD;
				  pT->m_sOutMsg.m_sbyFor  = DIR_101TOPH;
				  pT->m_sOutMsg.m_sbyType = DL_DATA_RES;
				  pMsg[byLen] = pT->CreateCRC(pT,&pMsg[4],pMsg[1]);
				  FPUT(DEV_RSMMD_BOX_ID,(BYTE*)&pT->m_sOutMsg);
			 break;
			 case EV_NACK_SC01_CON:
			 //case EV_ACK_RR08_RES:
				  byCMD = EV_NACK_SC01_CON;
				  memcpy(&pT->m_sOutMsg,pT->m_pOutMsg,pT->m_pOutMsg->m_swLen);
				  byLen = pMsg[1]+6-2;
				  pMsg[4]                 = (pB->v[DFC]<<4)|(pB->v[ACD]<<5)|byCMD;
				  pT->m_sOutMsg.m_sbyFor  = DIR_101TOPH;
				  pT->m_sOutMsg.m_sbyType = DL_DATA_RES;
				  pMsg[byLen] = pT->CreateCRC(pT,&pMsg[4],pMsg[1]);
				  FPUT(DEV_RSMMD_BOX_ID,(BYTE*)&pT->m_sOutMsg);
			 break;
			 case EV_NACK_RR08_RES:
				  FSMRB(BOX_L4);
				  //FSMRB(BOX_L4);
			 case EV_ACK_SC00_CON:
			 case EV_STJOIN_RR08_RES:
			      pMsg[0] = 0x10;
				  pMsg[1] = (pB->v[DFC]<<4)|(pB->v[ACD]<<5)|byMsgType;
				  pMsg[2] = pT->m_byModuleID;
				  pMsg[3] = pT->CreateCRC(pT,&pMsg[1],2);
				  pMsg[4] = 0x16;
				  pT->m_sOutMsg.m_swLen   = 9 + 5;
				  pT->m_sOutMsg.m_sbyFor  = DIR_101TOPH;
				  pT->m_sOutMsg.m_sbyType = DL_DATA_RES;
				  blSend = TRUE;
				  FPUT(DEV_RSMMD_BOX_ID,(BYTE*)&pT->m_sOutMsg);
			 break;
			 default:
			 break;
		   }
	  break;
	  case DIR_101TO101:
		   pT->m_sOutMsg.m_swLen        = 9;
		   pT->m_sOutMsg.m_sbyFrom      = byFor;
		   pT->m_sOutMsg.m_sbyFor       = byFor;
		   pT->m_sOutMsg.m_sbyIntType   = 0;
		   pT->m_sOutMsg.m_sbyServerID  = 0;
		   pT->m_sOutMsg.m_sbyType      = byMsgType;
		   pT->m_sOutMsg.m_sbyDirection = 0;
		   pT->m_sOutMsg.m_sbySensor    = 0;
		   FPUT(DEV_101MD_BOX_ID,(BYTE*)&pT->m_sOutMsg);
	  break;
	  case DIR_101TOKP:
		   switch(byMsgType)
		   {
		     case PH_CONN_IND:
			 case PH_DISC_IND:
				  pT->m_sOutMsg.m_swLen   = 9;
				  pT->m_sOutMsg.m_sbyFor  = DIR_101TOKP;
				  pT->m_sOutMsg.m_sbyType = byMsgType;
				  blSend = TRUE;
				  FPUT(DEV_KPMDL_BOX_ID,(BYTE*)&pT->m_sOutMsg);
		     break;
		     case PL_DATA_IND:
				  pT->m_sOutMsg.m_sbyFor  = DIR_101TOKP;
				  pT->m_sOutMsg.m_sbyType = PL_DATA_IND;
                  byAsduCode = pT->m_sOutMsg.m_sbyInfo[6];
				  switch(byAsduCode)
				  {
				    case MSG_TIME_ST_CODE:
						 pTME = (FTIME*)&pT->m_sOutMsg.m_sbyInfo[11];
						 pT->m_sOutMsg.m_sbyInfo[0]  = 11;
						 pT->m_sOutMsg.m_sbyInfo[1]  = pTME->IOA00;
						 pT->m_sOutMsg.m_sbyInfo[2]  = pTME->IOA01;
						 pT->m_sOutMsg.m_sbyInfo[3]  = pTME->IOA02;
						 pT->m_sOutMsg.m_sbyInfo[4]  = pTME->MSecL;
						 pT->m_sOutMsg.m_sbyInfo[5]  = pTME->MSecH;
						 pT->m_sOutMsg.m_sbyInfo[6]  = pTME->Min;
						 pT->m_sOutMsg.m_sbyInfo[7]  = pTME->Hour;
						 pT->m_sOutMsg.m_sbyInfo[8]  = pTME->DayM;
						 pT->m_sOutMsg.m_sbyInfo[9]  = pTME->Month;
						 pT->m_sOutMsg.m_sbyInfo[10] = pTME->Year;
						 pT->m_sOutMsg.m_swLen      = 9+pT->m_sOutMsg.m_sbyInfo[0];
						 blSend = TRUE;
						 FPUT(DEV_KPMDL_BOX_ID,(BYTE*)&pT->m_sOutMsg);
					break;
				    case PL_ASDU_DC0_IND:
						 pDCO = (FDCO*)&pT->m_sOutMsg.m_sbyInfo[11];
						 pT->m_sOutMsg.m_sbyInfo[0] = 6;
						 pT->m_sOutMsg.m_sbyInfo[1] = pDCO->IOA00;
						 pT->m_sOutMsg.m_sbyInfo[2] = pDCO->IOA01;
						 pT->m_sOutMsg.m_sbyInfo[3] = pDCO->IOA02;
						 pT->m_sOutMsg.m_sbyInfo[4] = 1;
						 pT->m_sOutMsg.m_sbyInfo[5] = (pDCO->DCS&0x0f)-1;
						 pT->m_sOutMsg.m_sbySensor  = pDCO->IOA00;
						 pT->m_sOutMsg.m_swLen      = 9+pT->m_sOutMsg.m_sbyInfo[0];
						 blSend = TRUE;
						 FPUT(DEV_KPMDL_BOX_ID,(BYTE*)&pT->m_sOutMsg);
					break;
				    case PL_ASDU_NVA_IND:
						 pNVA = (FNVA*)&pT->m_sOutMsg.m_sbyInfo[11];
						 pT->m_sOutMsg.m_sbyInfo[0] = 7;
						 pT->m_sOutMsg.m_sbyInfo[1] = pNVA->IOA00;
						 pT->m_sOutMsg.m_sbyInfo[2] = pNVA->IOA01;
						 pT->m_sOutMsg.m_sbyInfo[3] = pNVA->IOA02;
						 pT->m_sOutMsg.m_sbyInfo[4] = 2;
                         #ifdef WIN32
                         pT->m_sOutMsg.m_sbyInfo[5] = pNVA->byNvaL;
						 pT->m_sOutMsg.m_sbyInfo[6] = pNVA->byNvaH;
                         #else
                         pT->m_sOutMsg.m_sbyInfo[5] = pNVA->byNvaH;
						 pT->m_sOutMsg.m_sbyInfo[6] = pNVA->byNvaL;
                         #endif
						 pT->m_sOutMsg.m_swLen      = 9+pT->m_sOutMsg.m_sbyInfo[0];
						 blSend = TRUE;
						 FPUT(DEV_KPMDL_BOX_ID,(BYTE*)&pT->m_sOutMsg);
					break;
					default:
					break;
				  }
				  //pDCO = pT->m_sInMsg.m_sbyInfo[5];
				  //pT->m_sOutMsg.m_sbySensor= pT->m_sInMsg.m_sbyInfo[5];
				  //pT->m_sOutMsg.m_sbyDirection= pT->m_sInMsg.m_sbyInfo[6];

			 break;
			 default:
			 break;
		   }
	  break;
	  default:
	  break;
	}
	#ifdef DEB_C101Module
	if(blSend==TRUE)Info("\n(__)C101M::>OUTP::%M",&pT->m_sOutMsg);
	#endif
	return TRUE;
}
_GLOBAL SINT nADS;
BYTE CModule101_AddADSU(This,BYTE *pMsg,BYTE byNum)
{
    DECLARE_MULTI_OPEN(CModule101,CCyclicSystem)
	BYTE i,byLen,byNAdsu=0,byLenAdsu=sizeof(FTNVA),byLHead = sizeof(SADSUHEAD);
	SKPEVENT sEV;
	SADSUHEAD *pADH = (SADSUHEAD*)pMsg;
	FTNVA     *pNVA;
	pADH->Type     = 9;
	pADH->Cause    = 0x07;
	pADH->CAA00    = 2;
	pADH->CAA01    = 3;
	nADS++;
    for(i=0;i<byNum;i++)
	{
	if(FGET1(BOX_L4,(BYTE*)&sEV)!=0)
	{
	 #ifdef DEB_C101Module
	 Info("\n(__)C101M::>FGET::EV:Len:%b I::%b L::%b NA::%b LL::%w",&byNAdsu,&i,&byLenAdsu,&nADS,&sEV.wLen);
	 #endif
	 pNVA         = (FTNVA*)&pMsg[byLHead+byNAdsu];
	 //Addr
	 pNVA->IOA00  = sEV.byType;
	 pNVA->IOA01  = sEV.byAddr;
     pNVA->IOA02  = sEV.byCause;
	 //Value
	 pNVA->byNvaL = (BYTE)(sEV.wValue);
	 pNVA->byNvaH = ((BYTE)(sEV.wValue>>8))&0x7f;
	 //DQ
	 pNVA->byQDS  = 0;
	 //Time
	 pNVA->MSecL  = sEV.sTime.tMSecL;
	 pNVA->MSecH  = sEV.sTime.tMSecH;
	 pNVA->Min    = sEV.sTime.tMin;
	 //pNVA->Res1   = 0;
	 //pNVA->IV     = 0;
	 pNVA->Hour   = sEV.sTime.tHour;
	 //pNVA->Res2   = 0;
	 //pNVA->SU     = 0;
	 pNVA->DayM   = sEV.sTime.tDay;
	 pNVA->Month  = sEV.sTime.tMonth;
	 //pNVA->Res3   = 0;
	 pNVA->Year   = sEV.sTime.tYear;
	 //pNVA->Res4   = 0;
     byNAdsu      = (i+1)*byLenAdsu;
	}else
	{
	  //Info("\n BREAK;");
	  break;
	}
	}
	pADH->VSQ     = i;
	byLen = 6+byNAdsu;
	return byLen;
}
BYTE CModule101_AddADSU1(This,BYTE *pMsg,BYTE byNum)
{
    DECLARE_MULTI_OPEN(CModule101,CCyclicSystem)
	BYTE i,byLen,byNAdsu=0,byLenAdsu=sizeof(FTNVA),byLHead = sizeof(SADSUHEAD);
	SKPEVENT sEV;
	SADSUHEAD *pADH = (SADSUHEAD*)pMsg;
	FTNVA     *pNVA;
	pADH->Type     = 9;
	pADH->Cause    = 0x07;
	pADH->CAA00    = 2;
	pADH->CAA01    = 3;
	nADS++;
    for(i=0;i<byNum;i++)
	{
	if(FGET1(BOX_L4_1,(BYTE*)&sEV)!=0)
	{
	 #ifdef DEB_C101Module
	 Info("\n(__)C101M::>FGET1::EV:Len:%b I::%b L::%b NA::%b LL::%w",&byNAdsu,&i,&byLenAdsu,&nADS,&sEV.wLen);
	 #endif
	 pNVA         = (FTNVA*)&pMsg[byLHead+byNAdsu];
	 //Addr
	 pNVA->IOA00  = sEV.byType;
	 pNVA->IOA01  = sEV.byAddr;
     pNVA->IOA02  = sEV.byCause;
	 //Value
	 pNVA->byNvaL = (BYTE)(sEV.wValue);
	 pNVA->byNvaH = ((BYTE)(sEV.wValue>>8))&0x7f;
	 //DQ
	 pNVA->byQDS  = 0;
	 //Time
	 pNVA->MSecL  = sEV.sTime.tMSecL;
	 pNVA->MSecH  = sEV.sTime.tMSecH;
	 pNVA->Min    = sEV.sTime.tMin;
	 //pNVA->Res1   = 0;
	 //pNVA->IV     = 0;
	 pNVA->Hour   = sEV.sTime.tHour;
	 //pNVA->Res2   = 0;
	 //pNVA->SU     = 0;
	 pNVA->DayM   = sEV.sTime.tDay;
	 pNVA->Month  = sEV.sTime.tMonth;
	 //pNVA->Res3   = 0;
	 pNVA->Year   = sEV.sTime.tYear;
	 //pNVA->Res4   = 0;
     byNAdsu      = (i+1)*byLenAdsu;
	}else
	{
	  //Info("\n BREAK;");
	  break;
	}
	}
	pADH->VSQ     = i;
	byLen = 6+byNAdsu;
	return byLen;
}
BYTE CModule101_AddBroadADSU(This,BYTE *pMsg,SKPEVENT *pEV)
{
    DECLARE_MULTI_OPEN(CModule101,CCyclicSystem)
	BYTE byLen,byNAdsu=0,byLenAdsu=sizeof(FTNVA),byLHead = sizeof(SADSUHEAD);
	SKPEVENT sEV;
	SADSUHEAD *pADH = (SADSUHEAD*)pMsg;
	FTNVA     *pNVA;
	pADH->Type   = 9;
	pADH->Cause  = 0x07;
	pADH->CAA00  = 2;
	pADH->CAA01  = 3;

	pNVA         = (FTNVA*)&pMsg[byLHead];
	//Addr
	pNVA->IOA00  = pEV->byType;
	pNVA->IOA01  = pEV->byAddr;
    pNVA->IOA02  = pEV->byCause;
	//Value
	//#ifdef WIN32
	pNVA->byNvaL = (BYTE)(pEV->wValue);
	pNVA->byNvaH = ((BYTE)(pEV->wValue>>8))&0x7f;
	//#else
	//pNVA->byNvaH = (BYTE)(pEV->wValue);
	//pNVA->byNvaL = ((BYTE)(pEV->wValue>>8))&0x7f;
	//#endif
	//DQ
	pNVA->byQDS  = 0;
	//Time
	pNVA->MSecL  = pEV->sTime.tMSecL;
	pNVA->MSecH  = pEV->sTime.tMSecH;
	pNVA->Min    = pEV->sTime.tMin;
	//pNVA->Res1   = 0;
	//pNVA->IV     = 0;
	pNVA->Hour   = pEV->sTime.tHour;
	//pNVA->Res2   = 0;
	//pNVA->SU     = 0;
	pNVA->DayM   = pEV->sTime.tDay;
	pNVA->Month  = pEV->sTime.tMonth;
	//pNVA->Res3   = 0;
	pNVA->Year   = pEV->sTime.tYear;
	//pNVA->Res4   = 0;

	byNAdsu      = byLenAdsu;
	pADH->VSQ    = 1;
	byLen        = 6+byNAdsu;
	return byLen;
}
BYTE CModule101_AddAdsuTS(This,BYTE *pMsg,BYTE byNum)
{
    DECLARE_MULTI_OPEN(CModule101,CCyclicSystem)
	BYTE i,byLen,byNAdsu=0,byLenAdsu=sizeof(FSIQ),byLHead=sizeof(SADSUHEAD);
	SKPEVENT sTS;
	SADSUHEAD *pADH = (SADSUHEAD*)pMsg;
	FSIQ      *pSIQ;
	pADH->Type     = 2;
	pADH->VSQ      = byNum;
	pADH->Cause    = 7;
	//pADH->Ordinator= 0;
	pADH->CAA00    = 0;
	pADH->CAA01    = 0;
	for(i=0;i<byNum;i++)
	{
	if(FGET(BOX_L4,&sTS))
	{
	 #ifdef DEB_C101Module
	 Info("\n(__)C101M::>FGET::TS");
	 #endif
	 pSIQ           = (FSIQ*)&pMsg[byLHead+byNAdsu];
	 //SIA
	 pSIQ->IOA00    = sTS.byAddr;
	 pSIQ->IOA01    = 0;
	 pSIQ->IOA02    = 0;
	 //SIQ&DQ
	 pSIQ->SPI      = (BYTE)sTS.wValue;
	 pSIQ->RES      = 0;
	 pSIQ->BL       = 0;
	 pSIQ->SB       = 0;
	 pSIQ->NT       = 0;
	 pSIQ->IV       = 0;
	 //TIME
     pSIQ->MSecL    = sTS.sTime.tMSecL;
	 pSIQ->MSecH    = sTS.sTime.tMSecH;
	 pSIQ->Min      = sTS.sTime.tMin;
	 pSIQ->Rest     = 0;
	 pSIQ->IVt      = 0;
	 byNAdsu        = (i+1)*byLenAdsu;
	}else break;
	}
	byLen = 6+byNAdsu;
	return byLen;
}
BYTE CModule101_PackADSU(This,BYTE *pMsg)
{
    DECLARE_MULTI_OPEN(CModule101,CCyclicSystem)
	BYTE i,byLen,byNAdsu=0,byLenAdsu=sizeof(FNVA),byLHead = sizeof(SADSUHEAD);
	SREGPARAM sP;
	BYTE *pM = (BYTE*)&sP;
	BYTE *pD = (BYTE*)&sP.wParam;
	SADSUHEAD *pADH = (SADSUHEAD*)pMsg;
	FNVA      *pNVA;
	pADH->Type     = 9;
	pADH->VSQ      = FCHECK(BOX_REG);
	pADH->Cause    = 0x07;
	pADH->CAA00    = 0;
	pADH->CAA01    = 0;
    for(i=0;i<pADH->VSQ;i++)
	{
	if(FGET(BOX_REG,pM))
	{
	 #ifdef DEB_C101Module
	 Info("\n(__)C101M::>FGET::RG:%M",pM);
	 #endif
	 pNVA           = (FNVA*)&pMsg[byLHead+byNAdsu];
	 //Addr
	 pNVA->IOA00    = sP.byA0;
	 pNVA->IOA01    = sP.byA1;
     pNVA->IOA02    = sP.byA2;
	 //Value
	 #ifdef WIN32
	 pNVA->byNvaL   = pD[0];
	 pNVA->byNvaH   = pD[1];
	 pNVA->byNvaH  &= 0x7f;
	 #else
	 pNVA->byNvaL   = pD[1];
	 pNVA->byNvaH   = pD[0];
	 pNVA->byNvaH  &= 0x7f;
	 #endif
	 //DQ
	 pNVA->OV       = 0;
	 pNVA->RES      = 0;
	 pNVA->BL       = 0;
	 pNVA->SB       = 0;
	 pNVA->NT       = 0;
	 pNVA->IV       = 0;
	 byNAdsu        = (i+1)*byLenAdsu;
	}else break;
	}
	byLen = 6+byNAdsu;
	return byLen;
}
void CModule101_CopyW(This,PVOID pvDst,PVOID pvSrc)
{
    DECLARE_MULTI_OPEN(CModule101,CCyclicSystem)
	BYTE *pDS = (BYTE*)pvDst;
	BYTE *pSR = (BYTE*)pvSrc;
    #ifndef WIN32
	pDS[0] = pSR[1];
	pDS[1] = pSR[0];
    #else
	pDS[0] = pSR[0];
	pDS[1] = pSR[1];
    #endif
}
BYTE CModule101_CreateCRC(This,BYTE *pMsg,BYTE byLen)
{
    DECLARE_MULTI_OPEN(CModule101,CCyclicSystem)
	BYTE i,sum = 0;
	for(i=0;i<=byLen-1;i++)sum += pMsg[i];
	return sum;
}
void CModule101_CModule101(This)
{
    DECLARE_MULTI_OPEN(CModule101,CCyclicSystem)
	DECLARE_REGISTRATION(CModule101,Init)
	DECLARE_REGISTRATION(CModule101,LoLevelHandler)
	DECLARE_REGISTRATION(CModule101,HiLevelHandler)
	DECLARE_REGISTRATION(CModule101,SendMessage)
	DECLARE_REGISTRATION(CModule101,CreateCRC)
	DECLARE_REGISTRATION(CModule101,AddADSU)
	DECLARE_REGISTRATION(CModule101,AddADSU1)
	DECLARE_REGISTRATION(CModule101,PackADSU)
	DECLARE_REGISTRATION(CModule101,CopyW)
	DECLARE_REGISTRATION(CModule101,GetW)
	DECLARE_REGISTRATION(CModule101,SendBroadcast)
	DECLARE_REGISTRATION(CModule101,AddBroadADSU)
	DECLARE_REGISTRATION(CModule101,Autorisation)
	DECLARE_VIRTUAL_FUNC(CModule101,EventHandler)
	DECLARE_VIRTUAL_FUNC(CModule101,HandleTask)
	DECLARE_VIRTUAL_FUNC(CModule101,GetStateList)
}
void CModule101_DCModule101(This)
{
	DECLARE_MULTI_OPEN(CModule101,CCyclicSystem)
}
DECLARE_MULTI_CREATE(CModule101,CCyclicSystem)
```

#### bnrmysystem.c
```c
/********************************************************************
 * COPYRIGHT -- Kontora
 ********************************************************************
 * Program: bnrmain
 * File: bnrlsens.c
 * Author: Abramenya
 * Created: January 19, 2009
 *******************************************************************/

#include "bnrmysystem.h"
#include "bnrdirmodule.h"
#ifdef _DEFAULT_INCLUDES
 #include <AsDefault.h>
#endif
#ifdef WIN32
BOOL blStateConnecting = FALSE;
#endif
_GLOBAL INT iCSystemVal;
extern SSOFTSWITCHTABLE  nSoftSwitchTable;
void CSystem_CreateSystem(This,SHARDCOMPUTERTABLE *pTable)
{
     DECLARE_MULTI_OPEN(CSystem,CCyclicSystem)
	 #ifdef DEB_CSystem
	 Info("\n(__)CSYST::>Create System: %s",pTable->chProgrammVersion);
     #endif
	 FINIT();
	 pT->m_pAdmin         = NULL;
     pT->m_pComputer      = NULL;
	 pT->m_pObsModule     = NULL;
	 pT->m_byTcpConn      = FALSE;
	 pT->m_bySystemID     = pTable->bySystemID;
	 pB->SetBoxID(pB,DEV_SYSTM_BOX_ID);
	 iCSystemVal++;
	 pT->CreateSysBox(pT);
     pT->CreateComputer(pT,pTable);
	 pT->CreateAdmin(pT);
	 pT->CreateProc(pT);
	 pT->CreateObserveModule(pT,pTable,&nSoftSwitchTable);
     #ifdef WIN32
	 //CreateGetProc(pT);
     #endif
	 //pT->m_blSystemInitState = 0;
}
void CSystem_CreateComputer(This,SHARDCOMPUTERTABLE *pTable)
{
     DECLARE_MULTI_OPEN(CSystem,CCyclicSystem)
	 pT->m_pComputer = NULL;
     New(sizeof(CComputer),pT->m_pComputer);
	 InitObject(CComputer,pT->m_pComputer);
	 if(pT->m_pComputer!=NULL)
	 {
      pT->m_pComputer->Init(pT->m_pComputer,pTable);
	 }
}
void CSystem_CreateAdmin(This)
{
     DECLARE_MULTI_OPEN(CSystem,CCyclicSystem)
	 pT->m_pAdmin = NULL;
     New(sizeof(CAdmin),pT->m_pAdmin);
	 InitObject(CAdmin,pT->m_pAdmin);
	 if(pT->m_pAdmin!=NULL)
	 {
	  pT->m_pAdmin->SetSystemID(pT->m_pAdmin,pT->m_bySystemID);
	  pT->m_pAdmin->Init(pT->m_pAdmin);
	 }
}
void CSystem_CreateSysBox(This)
{
     DECLARE_MULTI_OPEN(CSystem,CCyclicSystem)
 	 //FDEFINE(DEV_SYSTM_BOX_ID,DEV_SYSTM_BOX_SZ);
	 FDEFINE(DEV_ADMIN_BOX_ID,DEV_ADMIN_BOX_SZ);
	 //FDEFINE(DEV_ARMOT_BOX_ID,DEV_ARMOT_BOX_SZ);
 	 //FDEFINE(DEV_ARMAD_BOX_ID,DEV_ARMAD_BOX_SZ);
}
/*
     CComVS0    *m_nCVS0;
     CComVS1    *m_nCVS1;
	 CTcpServer *m_nTCP;
*/

void CSystem_CreateObserveModule(This,SHARDCOMPUTERTABLE *pTable,SSOFTSWITCHTABLE *pSoftSwitchTable)
{

	 DECLARE_MULTI_OPEN(CSystem,CCyclicSystem)

	 /*
	 New(sizeof(CKpModule),pT->m_pObsModule);
     InitObject(CKpModule,pT->m_pObsModule);
	 pT->m_pObsModule->m_pComputer = pT->m_pComputer;
	 if(pT->m_pObsModule!=NULL)pT->m_pObsModule->Init(pT->m_pObsModule,pTable,pSoftSwitchTable);
	 FCREATE(pT->m_pObsModule->pBase,"KPProc",DEV_CJOB_ST_RESM,1);

	 New(sizeof(CModule101),pT->m_p101);
	 InitObject(CModule101,pT->m_p101);
	 if(pT->m_p101!=NULL)pT->m_p101->Init(pT->m_p101);
	 FCREATE(pT->m_p101->pBase,"M101Proc",DEV_CJOB_ST_RESM,1);
	 */
/*
SARMINTERFACE nARM0   = {0,DEV_ARM_PORT_COM232,DEV_ARM_RATE_57600,0,{0    ,    0},{  EVEN,  D_8,  S_1,  0}};
SARMINTERFACE nARM1   = {1,DEV_ARM_PORT_COM232,DEV_ARM_RATE_57600,0,{0    ,    0},{  EVEN,  D_8,  S_1,  0}};
SARMINTERFACE nARM2   = {2,DEV_ARM_PORT_COM232,DEV_ARM_RATE_57600,0,{0    ,    0},{  EVEN,  D_8,  S_1,  0}};

SARMINTERFACE nARMTCP = {3,DEV_ARM_PORT_TCP,DEV_ARM_RATE_57600,0,{20001   ,20002},{  192,  168,  1,  4},"192.168.1.4"};
SARMINTERFACE nARMUDP = {4,DEV_ARM_PORT_UDP,DEV_ARM_RATE_100MB,0,{20003   ,20004},{  192,  168,  1,  5},"192.168.1.5"};
*/

	 New(sizeof(CMsModule),pT->m_nMS);
	 InitObject(CMsModule,pT->m_nMS);
	 pT->m_nMS->m_pComputer = pT->m_pComputer;
	 if(pT->m_nMS!=NULL)pT->m_nMS->Init(pT->m_nMS,pTable,pSoftSwitchTable);
	 FCREATE(pT->m_nMS->pBase,"Measure",DEV_CJOB_ST_RESM,1);

	 New(sizeof(CComServer),pT->m_nCom);
     InitObject(CComServer,pT->m_nCom);
	 if(pT->m_nCom!=NULL)pT->m_nCom->Init(pT->m_nCom,pTable->pArmInterface[0]);
	 FCREATE(pT->m_nCom->pBase,"RsProc",DEV_CJOB_ST_RESM,1);

	 New(sizeof(CComVS0),pT->m_nCVS0);
	 InitObject(CComVS0,pT->m_nCVS0);
	 if(pT->m_nCVS0!=NULL)pT->m_nCVS0->Init(pT->m_nCVS0,pTable->pArmInterface[1]);
	 FCREATE(pT->m_nCVS0->pBase,"RsVS0Proc",DEV_CJOB_ST_RESM,1);

	 New(sizeof(CComVS1),pT->m_nCVS1);
	 InitObject(CComVS1,pT->m_nCVS1);
	 if(pT->m_nCVS1!=NULL)pT->m_nCVS1->Init(pT->m_nCVS1,pTable->pArmInterface[2]);
	 FCREATE(pT->m_nCVS1->pBase,"RsVS1Proc",DEV_CJOB_ST_RESM,1);

	 New(sizeof(CTcpServer),pT->m_nTCP);
	 InitObject(CTcpServer,pT->m_nTCP);
	 if(pT->m_nTCP!=NULL)pT->m_nTCP->Init(pT->m_nTCP,pTable->pArmInterface[3]);
	 FCREATE(pT->m_nTCP->pBase,"RsTCPProc",DEV_CJOB_ST_RESM,1);

}
void CSystem_CreateProc(This)
{
     DECLARE_MULTI_OPEN(CSystem,CCyclicSystem)
	 //FCREATE(pB                         ,"SystemProc" ,DEV_CJOB_ST_RESM,1);
	 FCREATE(pT->m_pAdmin->pBase        ,"AdminProc"  ,DEV_CJOB_ST_RESM,4);
}
/*
void CSystem_CyclicProc(This)
{
	 DECLARE_MULTI_OPEN(CSystem,CCyclicSystem)
	 pB->m_dwAmoutQuant++;
     #ifdef DEB_CSystem
	 if(dwFL&DEB_OUT_CYC_SYSTM)
	 Info("\n(%b)CSYST::>Cyclic Process.",&pB->m_dwAmoutQuant);
     #endif
 	 pB->GetMessage(pB);
}
*/
BOOL CSystem_EventHandler(This,SMESSAGE *pMsg)
{
	 DECLARE_MULTI_OPEN(CSystem,CCyclicSystem)
	 BOOL res = TRUE;
	 //CObserveModule *pOB;
	 //CDirectionModule *pD;
     BYTE byFrequency;
     #ifdef DEB_CSystem
	 if(dwFL&DEB_OUT_BOX_SYSTM)
	 Info("\n(%b)CSYST::>MSG::%M",&pMsg->m_sbyServerID,(BYTE*)pMsg);
	 #endif
	 switch (pMsg->m_sbyFor)
	 {
       case MDL_HCOMM:
	   case MDL_ADMIN:
            FPUT(DEV_ADMIN_BOX_ID,(BYTE*)pMsg);
	   break;
	   case MDL_SYSTM:
		   switch(pMsg->m_sbyType)
		   {
		     case EV_SYSTM_RESET_BOARD_IND:
                  #if MYSYSTEM_ID != 5
				  pD = pT->m_pObsModule->m_pDirectionModule[0];
				  pD->m_byDefSett = pMsg->m_sbyInfo[1];
				  pD->Serialize(pD,TRUE);
                  #endif
				  pT->m_pResetTimer.OnTimer(&pT->m_pResetTimer,T5SEC);
			 break;
			 case EV_SYSTM_RESET_TIM_BRD_IND:
				  //Info("\n(%w)CSYST::>Reset Board",&pT->m_bySystemID);
				  #ifndef WIN32
				  SYSreset(1, 1);
				  #endif
			 break;
		     case EV_SYSTM_INIT_OBS_REQ:
				  //Info("\n(%w)CSYST::>%M",&pT->m_bySystemID,(BYTE*)pMsg);
				  //pT->CreateObserveModule(pT,&nSoftSwitchTable);
				  pT->SendMessage(pT,MDL_ADMIN,EV_SYSTM_INIT_OBS_IND);
			 break;
		     case EV_SYSTM_CLOSE_INPOTRS_REQ:  //Закрыть все входные порты 	96
			 break;
		     case EV_SYSTM_OPEN_INPOTRS_REQ:   //Открыть все входные порты	97
			 break;
		     case EV_SYSTM_CLOSE_OUTPOTRS_REQ: //Закрыть все выходные порты	98
			 break;
		     case EV_SYSTM_OPEN_OUTPOTRS_REQ:  //Открыть все выходные порты	99
			 break;
		     case EV_SYSTM_STOP_JOB_REQ:       //Остановить задачу	100
				  if (pMsg->m_sbyInfo[1]==0)  pT->m_pObsModule->pBase->Stop(pT->m_pObsModule->pBase);               //Observe
				  if (pMsg->m_sbyInfo[1]==1)  pT->pBase->Stop(pT->pBase);                                                   //System
				  if (pMsg->m_sbyInfo[1]==2)  pT->m_pAdmin->pBase->Stop(pT->m_pAdmin->pBase);                               //Admin
			 break;
		     case EV_SYSTM_START_JOB_REQ:      //Запустить задачу	101
				  if (pMsg->m_sbyInfo[1]==0)  pT->m_pObsModule->pBase->Start(pT->m_pObsModule->pBase);               //Observe
				  if (pMsg->m_sbyInfo[1]==1)  pT->pBase->Start(pT->pBase);                                                   //System
				  if (pMsg->m_sbyInfo[1]==2)  pT->m_pAdmin->pBase->Start(pT->m_pAdmin->pBase);                               //Admin
			 break;
		     case EV_SYSTM_FREQ_JOB_REQ:       //Установить частоту вызова задачи	102
				  byFrequency = pMsg->m_sbyInfo[2];
				  if (pMsg->m_sbyInfo[1]==0)  pT->m_pObsModule->pBase->SetPeriod(pT->m_pObsModule->pBase,byFrequency);//Observe
				  if (pMsg->m_sbyInfo[1]==1)  pT->pBase->SetPeriod(pT->pBase,byFrequency);                                    //System
				  if (pMsg->m_sbyInfo[1]==2)  pT->m_pAdmin->pBase->SetPeriod(pT->m_pAdmin->pBase,byFrequency);                //Admin
			 break;
		     default:
			 break;
			}
	   break;
	   case MDL_PSENS:
	   case MDL_SENSR:
       case MDL_SSENS:
	   case MDL_DIRMD:
       case MDL_OBSRV:
		    pT->m_pObsModule->EventHandler(pT->m_pObsModule,pMsg);
	   break;
	   case MDL_COMPT:
	   break;
	   default:
	   break;
	 }
     return res;
}
BOOL CSystem_SendMessage(This,BYTE byFor,BYTE byType)
{
	 BOOL res = TRUE;
     DECLARE_MULTI_OPEN(CSystem,CCyclicSystem)
	 SHORTMESSAGE m_sSysMsg;
	 m_sSysMsg.m_swLen        = 9;
	 m_sSysMsg.m_sbyFrom      = MDL_SYSTM;
	 m_sSysMsg.m_sbyFor       = byFor;
	 m_sSysMsg.m_sbyIntType   = DEV_SYS_INTERFACE;
	 m_sSysMsg.m_sbyServerID  = pT->m_bySystemID;
	 m_sSysMsg.m_sbyType      = byType;
	 m_sSysMsg.m_sbyDirection = 0;
	 m_sSysMsg.m_sbySensor    = 0;
	 FPUT(DEV_SYSTM_BOX_ID,(BYTE*)&m_sSysMsg);
	 return res;
}
void CSystem_SendMsg(This,SMESSAGE *pMsg)
{
	 DECLARE_MULTI_OPEN(CSystem,CCyclicSystem)
	 /*
	 INT byMsg;
	 pT->m_sSysMsg.m_swLen        = 20;
	 pT->m_sSysMsg.m_sbyFrom      = MDL_SYSTM;
	 pT->m_sSysMsg.m_sbyFor       = MDL_ANOUT;
	 pT->m_sSysMsg.m_sbyIntType   = 0;
	 pT->m_sSysMsg.m_sbyServerID  = 0;
	 pT->m_sSysMsg.m_sbyType      = 23;
	 pT->m_sSysMsg.m_sbyDirection = 5;
	 pT->m_sSysMsg.m_sbySensor    = 4;
	 pT->m_sSysMsg.m_sbyInfo[0]++;
	 for(byMsg=1;byMsg<400;byMsg++)pT->m_sSysMsg.m_sbyInfo[byMsg] = byMsg;
	 FPUT(DEV_ARMOT_BOX_ID,(BYTE*)&pT->m_sSysMsg);
	 */
}
void CSystem_SwitchSystem(This,SSOFTSWITCHTABLE *pSoftSwitchTable)
{
     DECLARE_MULTI_OPEN(CSystem,CCyclicSystem)
}
void CSystem_CSystem(This)
{
     DECLARE_MULTI_OPEN(CSystem,CCyclicSystem)
	 DECLARE_REGISTRATION(CSystem,CreateSystem)
	 DECLARE_REGISTRATION(CSystem,CreateComputer)
	 DECLARE_REGISTRATION(CSystem,CreateAdmin)
	 DECLARE_REGISTRATION(CSystem,CreateSysBox)
	 DECLARE_REGISTRATION(CSystem,CreateObserveModule)
	 DECLARE_REGISTRATION(CSystem,SwitchSystem)
	 DECLARE_REGISTRATION(CSystem,CreateProc)
	 DECLARE_REGISTRATION(CSystem,SendMsg)
	 DECLARE_REGISTRATION(CSystem,SendMessage)
	 //DECLARE_VIRTUAL_FUNC(CSystem,CyclicProc)
	 DECLARE_VIRTUAL_FUNC(CSystem,EventHandler)
	 InitObject(CMTimer,&pT->m_pResetTimer);
 	 pT->m_pResetTimer.SetTimer(&pT->m_pResetTimer,MDL_SYSTM,MDL_SYSTM,EV_SYSTM_RESET_TIM_BRD_IND,0,0,DEV_SYSTM_BOX_ID);
}
void CSystem_DCSystem(This)
{
	DECLARE_MULTI_OPEN(CSystem,CCyclicSystem)
	DestroyObject(CComputer,pT->m_pComputer);
	DestroyObject(CAdmin,pT->m_pAdmin);
    #if MYSYSTEM_ID != 5
	DestroyObject(CObserveModule,pT->m_pObsModule);
    #else
    #endif
	FDELETE(DEV_SYSTM_BOX_ID);
	FDELETE(DEV_ADMIN_BOX_ID);
	FDELETE(DEV_ARMOT_BOX_ID);
 	FDELETE(DEV_ARMAD_BOX_ID);
}
DECLARE_MULTI_CREATE(CSystem,CCyclicSystem)
#ifdef WIN32
SLMESSAGE sMSG;
SLMESSAGE gMSG;
INT ret;
WSADATA       wsd;
SOCKET        sClient1;
char          szBuffer[255];
char          szServer[255];
int           i;
struct sockaddr_in server;
struct hostent    *host = NULL;
DWORD dwTic;
DWORD WINAPI GetArmToSyst(PVOID pVoid)
{
	while(1)
	{
		ret = recv(sClient1, (BYTE*)&gMSG,sizeof(SLMESSAGE) , 0);
		if((ret!=0)&&(blStateConnecting)&&(ret != SOCKET_ERROR))
		{
		 //Info("\n(__)GET_SYS::%M",(BYTE*)&gMSG);
		 //printf("\n(%d)GET_SYS::%d",gMSG.m_swLen,gMSG.m_sbyType);
		 FPUT(DEV_SYSTM_BOX_ID,(BYTE*)&gMSG);
		}//else Sleep(10);
	}
	return 0;
}
DWORD WINAPI SendToArm(PVOID pVoid)
{
//	BYTE i;
//	SMESSAGE *pS;
//  BYTE *pM;
	while(1)
	{
		if(FGET(DEV_ARMOT_BOX_ID,(BYTE*)&sMSG)!=0)
		{
			//pS = &sMSG;
			//pM = (BYTE*)pS;
			//printf("\nOMSG::>");
			//for(i=0;i<pS->m_swLen;i++)printf(" %x",pM[i]);
			//Info("\n(__)PUT_ARM::%M",(BYTE*)&sMSG);
            //printf("\n(%d)PUT_ARM::%d",gMSG.m_swLen,sMSG.m_sbyType);
			ret = send(sClient1, (BYTE*)&sMSG, sMSG.m_swLen,  0);
		}//else
		Sleep(50);
		///////////////////////////////////////
        if(dwTic++%20==0)
		{
		  if(blStateConnecting==FALSE)
			if (connect(sClient1, (struct sockaddr *)&server, sizeof(server)) == SOCKET_ERROR)
			{
		 	 printf("\n(%d)Query connection",dwTic);
			 blStateConnecting = FALSE;
			}else
			{
				printf("\n(%d)Connection complette.",dwTic);
				blStateConnecting = TRUE;

			}
		}
		///////////////////////////////////////
	}
	return 0;
}
void CreateGetProc(PVOID pVD)
{
	DWORD dwThreadId, dwThrdParam = 1;
	HANDLE hThread;
    if (WSAStartup(MAKEWORD(2,2), &wsd) != 0)
    {
        printf("Failed to load Winsock library!\n");
        return ;
    }
    sClient1 = socket(AF_INET, SOCK_STREAM, IPPROTO_TCP);
    if (sClient1 == INVALID_SOCKET)
    {
        printf("socket() failed: %d\n", WSAGetLastError());
        return ;
    }
    server.sin_family = AF_INET;
    server.sin_port = htons(20010);
    server.sin_addr.s_addr = inet_addr("127.0.0.2");
    if (server.sin_addr.s_addr == INADDR_NONE)
    {
        host = gethostbyname(szServer);
        if (host == NULL)
        {
            printf("Unable to resolve server: %s\n", szServer);
            return ;
        }
        CopyMemory(&server.sin_addr, host->h_addr_list[0],host->h_length);
    }
	blStateConnecting = TRUE;
    if (connect(sClient1, (struct sockaddr *)&server, sizeof(server)) == SOCKET_ERROR)
    {
        printf("\nconnect() failed: %d", WSAGetLastError());
		blStateConnecting = FALSE;
    }else
	{
		printf("\n(%d)Connection complette.",dwTic);
		blStateConnecting = TRUE;
	}
	hThread = CreateThread(NULL,0,GetArmToSyst    ,pVD,0,&dwThreadId);
	hThread = CreateThread(NULL,0,SendToArm,pVD,0,&dwThreadId);
}
#endif
```
